# B&R Automation Studio project NAEUL004C00R13L518F00 (part 25)

#### Act_OptP1024Save.st
```iecst
ACTION Act_OptP1024Save:

	IF tyP1024McSetAntiGap.tyAntiGap.tyNumLftSenOff.bRtCompl
		OR tyP1024McSetAntiGap.tyAntiGap.tyNumMidSenOff.bRtCompl
		OR tyP1024McSetAntiGap.tyAntiGap.tyNumRgtSenOff.bRtCompl
		OR tyP1024McSetAntiGap.tyAntiGap.tyNumClrSenOff.bRtCompl
		OR tyP1024McSetAntiGap.tyAntiGap.tyNumMagConvEntOn.bRtCompl
		OR tyP1024McSetAntiGap.tyAntiGap.tyNumMagConvEntOff.bRtCompl
		OR tyP1024McSetAntiGap.tyAntiGap.tyNumMagConvPresentOn.bRtCompl
		OR tyP1024McSetAntiGap.tyAntiGap.tyNumMagConvPresentOff.bRtCompl
		THEN

		fUIInRtStatHide(ADR(tyCommon.tySet.tyBtnSave.uiMaskRtStat));

		tyP1024McSetAntiGap.tyAntiGap.tyNumLftSenOff.bRtCompl			:= FALSE;
		tyP1024McSetAntiGap.tyAntiGap.tyNumMidSenOff.bRtCompl			:= FALSE;
		tyP1024McSetAntiGap.tyAntiGap.tyNumRgtSenOff.bRtCompl			:= FALSE;
		tyP1024McSetAntiGap.tyAntiGap.tyNumClrSenOff.bRtCompl			:= FALSE;
		tyP1024McSetAntiGap.tyAntiGap.tyNumMagConvEntOn.bRtCompl		:= FALSE;
		tyP1024McSetAntiGap.tyAntiGap.tyNumMagConvEntOff.bRtCompl		:= FALSE;
		tyP1024McSetAntiGap.tyAntiGap.tyNumMagConvPresentOn.bRtCompl	:= FALSE;
		tyP1024McSetAntiGap.tyAntiGap.tyNumMagConvPresentOff.bRtCompl	:= FALSE;

	END_IF

	IF tyCommon.tySet.tyBtnSave.bRtCompl = TRUE THEN

		tyMcParamWr.tyLftSenAntiGapDly.diSigOffTm			:=  tyP1024McSetAntiGap.tyAntiGap.tyNumLftSenOff.diValue;
		tyMcParamWr.tyMidSenAntiGapDly.diSigOffTm			:=  tyP1024McSetAntiGap.tyAntiGap.tyNumMidSenOff.diValue;
		tyMcParamWr.tyRgtSenAntiGapDly.diSigOffTm			:=	tyP1024McSetAntiGap.tyAntiGap.tyNumRgtSenOff.diValue;
		tyMcParamWr.tyClrSenAntiGapDly.diSigOffTm			:=  tyP1024McSetAntiGap.tyAntiGap.tyNumClrSenOff.diValue;
		tyMcParamWr.tyMagConvEntrySenAntiGapDly.diSigOnTm	:=  tyP1024McSetAntiGap.tyAntiGap.tyNumMagConvEntOn.diValue;
		tyMcParamWr.tyMagConvEntrySenAntiGapDly.diSigOffTm	:=  tyP1024McSetAntiGap.tyAntiGap.tyNumMagConvEntOff.diValue;
		tyMcParamWr.tyMagConvPresentSenAntiGapDly.diSigOnTm	:=	tyP1024McSetAntiGap.tyAntiGap.tyNumMagConvPresentOn.diValue;
		tyMcParamWr.tyMagConvPresentSenAntiGapDly.diSigOffTm:=	tyP1024McSetAntiGap.tyAntiGap.tyNumMagConvPresentOff.diValue;

		eMcParamAct	:= McParamActWrite;

		IF p_eMcParamStat = McParamActWrite AND p_eMcParamStatus = Done THEN

			eMcParamAct	:= McParamActIdle;

			//Update BackUp Param
			tyP1024McSetAntiGap.tyAntiGapBkUp	:= tyP1024McSetAntiGap.tyAntiGap;

			tyCommon.tySet.tyBtnSave.bRtCompl 	:= FALSE;
			fUIInRtStatOff(ADR(tyCommon.tySet.tyBtnSave.uiMaskRtStat));

		ELSIF p_eMcParamStatus = Error THEN
			p_tyC0008MsgBox ACCESS ADR(tyP1024McSetAntiGap.tyMsgBoxSaveErr);

			IF tyP1024McSetAntiGap.tyMsgBoxSaveErr.tyBtnNo.bRtCompl = TRUE THEN
				tyP1024McSetAntiGap.tyMsgBoxSaveErr.tyBtnNo.bRtCompl	:= FALSE;
				tyP1024McSetAntiGap.tyMsgBoxSaveErr.tyBtnNo.bValue		:= FALSE;

				p_tyC0008MsgBox ACCESS ADR(tyP1024McSetAntiGap.tyMsgBoxHide);

				//Restore Param
				tyP1024McSetAntiGap.tyAntiGap	:= tyP1024McSetAntiGap.tyAntiGapBkUp;
				tyMcParamWr						:= p_tyMcParamCurr;

				tyCommon.tySet.tyBtnSave.bRtCompl 	:= FALSE;
				fUIInRtStatOff(ADR(tyCommon.tySet.tyBtnSave.uiMaskRtStat));
			END_IF

		END_IF

	END_IF

END_ACTION
```

#### Act_OptP1024Keypad.st
```iecst
ACTION Act_OptP1024Keypad:

	IF fUIOutRtStatTPIsOpen(ADR(tyP1024McSetAntiGap.tyAntiGap.tyNumLftSenOff.uiRtStat)) = TRUE THEN
		tyProperty.tyKeypad.tyStringTitle.sKeypadTitle	:= tyP1024McSetAntiGap.tyAntiGap.tyNumLftSenOff.sKeypadTitle;

	ELSIF fUIOutRtStatTPIsOpen(ADR(tyP1024McSetAntiGap.tyAntiGap.tyNumMidSenOff.uiRtStat)) = TRUE THEN
		tyProperty.tyKeypad.tyStringTitle.sKeypadTitle	:= tyP1024McSetAntiGap.tyAntiGap.tyNumMidSenOff.sKeypadTitle;

	ELSIF fUIOutRtStatTPIsOpen(ADR(tyP1024McSetAntiGap.tyAntiGap.tyNumRgtSenOff.uiRtStat)) = TRUE THEN
		tyProperty.tyKeypad.tyStringTitle.sKeypadTitle	:= tyP1024McSetAntiGap.tyAntiGap.tyNumRgtSenOff.sKeypadTitle;

	ELSIF fUIOutRtStatTPIsOpen(ADR(tyP1024McSetAntiGap.tyAntiGap.tyNumClrSenOff.uiRtStat)) = TRUE THEN
		tyProperty.tyKeypad.tyStringTitle.sKeypadTitle	:= tyP1024McSetAntiGap.tyAntiGap.tyNumClrSenOff.sKeypadTitle;

	ELSIF fUIOutRtStatTPIsOpen(ADR(tyP1024McSetAntiGap.tyAntiGap.tyNumMagConvEntOff.uiRtStat)) = TRUE THEN
		tyProperty.tyKeypad.tyStringTitle.sKeypadTitle	:= tyP1024McSetAntiGap.tyAntiGap.tyNumMagConvEntOff.sKeypadTitle;

	ELSIF fUIOutRtStatTPIsOpen(ADR(tyP1024McSetAntiGap.tyAntiGap.tyNumMagConvEntOn.uiRtStat)) = TRUE THEN
		tyProperty.tyKeypad.tyStringTitle.sKeypadTitle	:= tyP1024McSetAntiGap.tyAntiGap.tyNumMagConvEntOn.sKeypadTitle;

	ELSIF fUIOutRtStatTPIsOpen(ADR(tyP1024McSetAntiGap.tyAntiGap.tyNumMagConvPresentOff.uiRtStat)) = TRUE THEN
		tyProperty.tyKeypad.tyStringTitle.sKeypadTitle	:= tyP1024McSetAntiGap.tyAntiGap.tyNumMagConvEntOn.sKeypadTitle;

	ELSIF fUIOutRtStatTPIsOpen(ADR(tyP1024McSetAntiGap.tyAntiGap.tyNumMagConvPresentOn.uiRtStat)) = TRUE THEN
		tyProperty.tyKeypad.tyStringTitle.sKeypadTitle	:= tyP1024McSetAntiGap.tyAntiGap.tyNumMagConvEntOn.sKeypadTitle;

	END_IF

END_ACTION
```

#### Act_EntP1025Disp.st
```iecst
ACTION Act_EntP1025Disp:

	//Access Address
	p_tyC0004Navi ACCESS ADR(tyP1025McSetScan.tyNaviBack);

	p_tyC0005Main ACCESS ADR(tyCommon.tyMain);

	p_tyC0006Set ACCESS ADR(tyCommon.tySet);

	p_tyC0007Notif ACCESS ADR(tyCommon.tyNotif);

	p_tyC0008MsgBox ACCESS ADR (tyP1025McSetScan.tyMsgBoxHide);

	p_tyC0009Info ACCESS ADR(tyCommon.tyInfo);

	p_tyP1025McSetScan ACCESS ADR(tyP1025McSetScan.tyScan);

	//Backup Param
	tyP1025McSetScan.tyScanBkUp	:= tyP1025McSetScan.tyScan;

END_ACTION
```

#### Act_ExitP1025.st
```iecst
ACTION Act_ExitP1025:

	IF tyCommon.tySet.tyBtnSave.uiMaskRtStat.0 = FALSE THEN
		usiChgPage	:= 1;

	ELSE

		p_tyC0008MsgBox ACCESS ADR(tyP1025McSetScan.tyMsgBoxExitAsk);

		IF tyP1025McSetScan.tyMsgBoxExitAsk.tyBtnYes.bRtCompl = TRUE THEN
			tyP1025McSetScan.tyMsgBoxExitAsk.tyBtnYes.bRtCompl	:= FALSE;
			tyP1025McSetScan.tyMsgBoxExitAsk.tyBtnYes.bValue		:= FALSE;

			p_tyC0008MsgBox ACCESS ADR(tyP1025McSetScan.tyMsgBoxHide);

			//Restore Param
			tyP1025McSetScan.tyScan	:= tyP1025McSetScan.tyScanBkUp;

			fUIInRtStatOff(ADR(tyCommon.tySet.tyBtnSave.uiMaskRtStat));

			usiChgPage	:= 1;

		ELSIF tyP1025McSetScan.tyMsgBoxExitAsk.tyBtnNo.bRtCompl = TRUE THEN
			tyP1025McSetScan.tyMsgBoxExitAsk.tyBtnNo.bRtCompl	:= FALSE;
			tyP1025McSetScan.tyMsgBoxExitAsk.tyBtnNo.bValue		:= FALSE;

			p_tyC0008MsgBox ACCESS ADR(tyP1025McSetScan.tyMsgBoxHide);

			eChgPage	:= eCurrPage;
			usiChgPage	:= 0;

		END_IF

	END_IF

END_ACTION
```

#### Act_OptP1025Navi.st
```iecst
ACTION Act_OptP1025Navi:

	tyP1025McSetScan.tyNaviBack.tyBtnBack.bRtLk	:= tyCommon.tySet.tyBtnSave.bRtCompl;

	IF tyP1025McSetScan.tyNaviBack.tyBtnBack.bRtCompl = TRUE THEN
		tyP1025McSetScan.tyNaviBack.tyBtnBack.bRtCompl	:= FALSE;

		eChgPage	:= UIP1020McSetNavi;

	END_IF

END_ACTION
```

#### Act_OptP1025Save.st
```iecst
ACTION Act_OptP1025Save:

	IF tyP1025McSetScan.tyScan.tyStringTopScanSvrIP.bRtCompl OR tyP1025McSetScan.tyScan.tyNumTopScanSvrPort.bRtCompl
		OR tyP1025McSetScan.tyScan.tyStringTopScanSvrIP.bRtCompl OR tyP1025McSetScan.tyScan.tyNumBtmScanSvrPort.bRtCompl
		OR tyP1025McSetScan.tyScan.tyBtnTopScanEn.bRtCompl OR tyP1025McSetScan.tyScan.tyBtnBtmScanEn.bRtCompl THEN

		fUIInRtStatHide(ADR(tyCommon.tySet.tyBtnSave.uiMaskRtStat));

		tyP1025McSetScan.tyScan.tyStringTopScanSvrIP.bRtCompl			:= FALSE;
		tyP1025McSetScan.tyScan.tyNumTopScanSvrPort.bRtCompl			:= FALSE;
		tyP1025McSetScan.tyScan.tyStringTopScanSvrIP.bRtCompl			:= FALSE;
		tyP1025McSetScan.tyScan.tyNumBtmScanSvrPort.bRtCompl			:= FALSE;
		tyP1025McSetScan.tyScan.tyBtnTopScanEn.bRtCompl					:= FALSE;
		tyP1025McSetScan.tyScan.tyBtnBtmScanEn.bRtCompl					:= FALSE;

	END_IF

	IF tyCommon.tySet.tyBtnSave.bRtCompl = TRUE THEN

		tyMcParamWr.sTopScanIPAddr			:=  tyP1025McSetScan.tyScan.tyStringTopScanSvrIP.sValue;
		tyMcParamWr.uiTopScanSvrPort		:=  DINT_TO_UINT (tyP1025McSetScan.tyScan.tyNumTopScanSvrPort.diValue);
		tyMcParamWr.sBtmScanIPAddr			:=	tyP1025McSetScan.tyScan.tyStringBtmScanSvrIP.sValue;
		tyMcParamWr.uiBtmScanSvrPort		:=  DINT_TO_UINT (tyP1025McSetScan.tyScan.tyNumBtmScanSvrPort.diValue);
		tyMcParamWr.bTopScannerEn			:=  tyP1025McSetScan.tyScan.tyBtnTopScanEn.bValue;
		tyMcParamWr.bBtmScannerEn			:=  tyP1025McSetScan.tyScan.tyBtnBtmScanEn.bValue;

		eMcParamAct	:= McParamActWrite;

		IF p_eMcParamStat = McParamActWrite AND p_eMcParamStatus = Done THEN

			eMcParamAct	:= McParamActIdle;

			//Update BackUp Param
			tyP1025McSetScan.tyScanBkUp	:= tyP1025McSetScan.tyScan;

			tyCommon.tySet.tyBtnSave.bRtCompl 	:= FALSE;
			fUIInRtStatOff(ADR(tyCommon.tySet.tyBtnSave.uiMaskRtStat));

		ELSIF p_eMcParamStatus = Error THEN
			p_tyC0008MsgBox ACCESS ADR(tyP1025McSetScan.tyMsgBoxSaveErr);

			IF tyP1025McSetScan.tyMsgBoxSaveErr.tyBtnNo.bRtCompl = TRUE THEN
				tyP1025McSetScan.tyMsgBoxSaveErr.tyBtnNo.bRtCompl	:= FALSE;
				tyP1025McSetScan.tyMsgBoxSaveErr.tyBtnNo.bValue		:= FALSE;

				p_tyC0008MsgBox ACCESS ADR(tyP1025McSetScan.tyMsgBoxHide);

				//Restore Param
				tyP1025McSetScan.tyScan	:= tyP1025McSetScan.tyScanBkUp;
				tyMcParamWr						:= p_tyMcParamCurr;

				tyCommon.tySet.tyBtnSave.bRtCompl 	:= FALSE;
				fUIInRtStatOff(ADR(tyCommon.tySet.tyBtnSave.uiMaskRtStat));
			END_IF

		END_IF

	END_IF

END_ACTION
```

#### Act_OptP1025Keypad.st
```iecst
ACTION Act_OptP1025Keypad:

	IF fUIOutRtStatTPIsOpen(ADR(tyP1025McSetScan.tyScan.tyStringTopScanSvrIP.uiRtStat)) = TRUE THEN
		tyProperty.tyKeypad.tyStringTitle.sKeypadTitle	:= tyP1025McSetScan.tyScan.tyStringTopScanSvrIP.sKeypadTitle;

	ELSIF fUIOutRtStatTPIsOpen(ADR(tyP1025McSetScan.tyScan.tyNumTopScanSvrPort.uiRtStat)) = TRUE THEN
		tyProperty.tyKeypad.tyStringTitle.sKeypadTitle	:= tyP1025McSetScan.tyScan.tyNumTopScanSvrPort.sKeypadTitle;

	ELSIF fUIOutRtStatTPIsOpen(ADR(tyP1025McSetScan.tyScan.tyStringBtmScanSvrIP.uiRtStat)) = TRUE THEN
		tyProperty.tyKeypad.tyStringTitle.sKeypadTitle	:= tyP1025McSetScan.tyScan.tyStringBtmScanSvrIP.sKeypadTitle;

	ELSIF fUIOutRtStatTPIsOpen(ADR(tyP1025McSetScan.tyScan.tyNumBtmScanSvrPort.uiRtStat)) = TRUE THEN
		tyProperty.tyKeypad.tyStringTitle.sKeypadTitle	:= tyP1025McSetScan.tyScan.tyNumBtmScanSvrPort.sKeypadTitle;

	END_IF

END_ACTION
```

#### Act_EntP1026Disp.st
```iecst
ACTION Act_EntP1026Disp:

	//Access Address
	p_tyC0002FullMask ACCESS ADR(tyP1026McSetTeach.tyFullMaskHide);

	p_tyC0004Navi ACCESS ADR(tyP1026McSetTeach.tyNaviBack);

	p_tyC0005Main ACCESS ADR(tyCommon.tyMain);

	p_tyC0007Notif ACCESS ADR(tyCommon.tyNotif);

	p_tyC0008MsgBox ACCESS ADR(tyP1026McSetTeach.tyMsgBoxHide);

	p_tyC0009Info ACCESS ADR(tyCommon.tyInfo);

	p_tyP1026InOutletShutterFB ACCESS ADR(tyP1026McSetTeach.tyInOutletShutterFB);

	IF bTeachTravPosA = TRUE THEN
		p_tyP1026McSetTeach ACCESS ADR(tyP1026McSetTeach.tyTeachTravPosA);
		p_tyC0001MotionStd ACCESS ADR(tyP1026McSetTeach.tyMotionStdTrav);

	ELSIF bTeachTravPosB = TRUE THEN
		p_tyP1026McSetTeach ACCESS ADR(tyP1026McSetTeach.tyTeachTravPosB);
		p_tyC0001MotionStd ACCESS ADR(tyP1026McSetTeach.tyMotionStdTrav);

	ELSIF bTeachLifterPosA = TRUE THEN
		p_tyP1026McSetTeach ACCESS ADR(tyP1026McSetTeach.tyTeachLifterPosA);
		p_tyC0001MotionStd ACCESS ADR(tyP1026McSetTeach.tyMotionStdLifter);

	ELSIF bTeachLifterPosB = TRUE THEN
		p_tyP1026McSetTeach ACCESS ADR(tyP1026McSetTeach.tyTeachLifterPosB);
		p_tyC0001MotionStd ACCESS ADR(tyP1026McSetTeach.tyMotionStdLifter);

	ELSIF bTeachLifterTopPos THEN
		p_tyP1026McSetTeach ACCESS ADR(tyP1026McSetTeach.tyTeachLifterTopPos);
		p_tyC0001MotionStd ACCESS ADR(tyP1026McSetTeach.tyMotionStdLifter);

	ELSIF bTeachLifterBtmPos THEN
		p_tyP1026McSetTeach ACCESS ADR(tyP1026McSetTeach.tyTeachLifterBtmPos);
		p_tyC0001MotionStd ACCESS ADR(tyP1026McSetTeach.tyMotionStdLifter);

	ELSIF bTeachLifterTopPos2 THEN
		p_tyP1026McSetTeach ACCESS ADR(tyP1026McSetTeach.tyTeachLifterTopPos2);
		p_tyC0001MotionStd ACCESS ADR(tyP1026McSetTeach.tyMotionStdLifter); //Lifter2FBCtrl

	ELSIF bTeachLifterBtmPos2 THEN
		p_tyP1026McSetTeach ACCESS ADR(tyP1026McSetTeach.tyTeachLifterBtmPos2);
		p_tyC0001MotionStd ACCESS ADR(tyP1026McSetTeach.tyMotionStdLifter);

	END_IF

	//Display
	//Traverser
	tyP1026McSetTeach.tyMotionStdTrav.tyBtnPwr.bValue	:= p_bTravPwrOn;

	//Lifter
	tyP1026McSetTeach.tyMotionStdLifter.tyBtnPwr.bValue	:= p_bLifterBtmPwrOn;

END_ACTION
```

#### Act_ExitP1026.st
```iecst
ACTION Act_ExitP1026:

	usiChgPage	:= 1;

	//Manual Deactivated
	bManualMod	:= FALSE;

	//Reset UI
	bJogSlow				:= FALSE;
	bJogFast				:= FALSE;
	fbJogSlowToFastDlyTm.IN	:= FALSE;

	fbLmtRstTm(IN := FALSE);
	//bypass curtain sensor
	bBypCurtainSen := FALSE;
	bBypCurtainPBLED := FALSE;
	tyP1026McSetTeach.tyTeachTravPosA.tyBtn4.bValue				:= FALSE;
	tyP1026McSetTeach.tyTeachTravPosB.tyBtn4.bValue				:= FALSE;
	tyP1026McSetTeach.tyTeachLifterPosA.tyBtn4.bValue				:= FALSE;
	tyP1026McSetTeach.tyTeachLifterPosB.tyBtn4.bValue				:= FALSE;

	//Traverser
	tyP1026McSetTeach.tyMotionStdTrav.tyBtnPwr.bRtCompl				:= FALSE;
	tyP1026McSetTeach.tyMotionStdTrav.tyBtnStop.bRtCompl			:= FALSE;
	tyP1026McSetTeach.tyMotionStdTrav.tyBtnOrigin.bRtCompl			:= FALSE;
	tyP1026McSetTeach.tyMotionStdTrav.tyBtnRst.bRtCompl				:= FALSE;
	tyP1026McSetTeach.tyMotionStdTrav.tyBtnMovAbs.bRtCompl			:= FALSE;
	tyP1026McSetTeach.tyMotionStdTrav.tyBtnMovRel.bRtCompl			:= FALSE;
	tyP1026McSetTeach.tyMotionStdTrav.tyBtnJogFront.bRtCompl		:= FALSE;
	tyP1026McSetTeach.tyMotionStdTrav.tyBtnJogRear.bRtCompl			:= FALSE;

	tyP1026McSetTeach.tyTeachTravPosA.tyBtn2.bRtCompl				:= FALSE;
	tyP1026McSetTeach.tyTeachTravPosB.tyBtn2.bRtCompl				:= FALSE;

	tyP1026McSetTeach.tyMotionStdTrav.tyBtnPwr.bValue				:= FALSE;
	tyP1026McSetTeach.tyMotionStdTrav.tyBtnStop.bValue				:= TRUE;
	tyP1026McSetTeach.tyMotionStdTrav.tyBtnOrigin.bValue			:= FALSE;
	tyP1026McSetTeach.tyMotionStdTrav.tyBtnRst.bValue				:= FALSE;
	tyP1026McSetTeach.tyMotionStdTrav.tyBtnMovAbs.bValue			:= FALSE;
	tyP1026McSetTeach.tyMotionStdTrav.tyBtnMovRel.bValue			:= FALSE;
	tyP1026McSetTeach.tyMotionStdTrav.tyBtnJogFront.bValue			:= FALSE;
	tyP1026McSetTeach.tyMotionStdTrav.tyBtnJogRear.bValue			:= FALSE;

	tyP1026McSetTeach.tyTeachTravPosA.tyBtn2.bValue					:= FALSE;
	tyP1026McSetTeach.tyTeachTravPosB.tyBtn2.bValue					:= FALSE;

	tyP1026McSetTeach.tyMotionStdTrav.tyBtnPwr.bRtLk				:= FALSE;
	tyP1026McSetTeach.tyMotionStdTrav.tyBtnStop.bRtLk				:= TRUE;
	tyP1026McSetTeach.tyMotionStdTrav.tyBtnOrigin.bRtLk				:= FALSE;
	tyP1026McSetTeach.tyMotionStdTrav.tyBtnRst.bRtLk				:= FALSE;
	tyP1026McSetTeach.tyMotionStdTrav.tyBtnMovAbs.bRtLk				:= FALSE;
	tyP1026McSetTeach.tyMotionStdTrav.tyBtnMovRel.bRtLk				:= FALSE;
	tyP1026McSetTeach.tyMotionStdTrav.tyBtnJogFront.bRtLk			:= FALSE;
	tyP1026McSetTeach.tyMotionStdTrav.tyBtnJogRear.bRtLk			:= FALSE;

	tyP1026McSetTeach.tyTeachTravPosA.tyBtn2.bRtLk					:= FALSE;
	tyP1026McSetTeach.tyTeachTravPosB.tyBtn2.bRtLk					:= FALSE;

	tyP1026McSetTeach.tyMotionStdTrav.tyBtnPwr.uiMaskRtStat			:= TRUE;
	tyP1026McSetTeach.tyMotionStdTrav.tyBtnOrigin.uiMaskRtStat		:= FALSE;
	tyP1026McSetTeach.tyMotionStdTrav.tyBtnRst.uiMaskRtStat			:= TRUE;
	tyP1026McSetTeach.tyMotionStdTrav.tyBtnMovAbs.uiMaskRtStat		:= FALSE;
	tyP1026McSetTeach.tyMotionStdTrav.tyBtnMovRel.uiMaskRtStat		:= FALSE;
	tyP1026McSetTeach.tyMotionStdTrav.tyBtnJogFront.uiMaskRtStat	:= FALSE;
	tyP1026McSetTeach.tyMotionStdTrav.tyBtnJogRear.uiMaskRtStat		:= FALSE;

	tyP1026McSetTeach.tyTeachTravPosA.tyBtn2.uiMaskRtStat			:= FALSE;
	tyP1026McSetTeach.tyTeachTravPosB.tyBtn2.uiMaskRtStat			:= FALSE;

	//Lifter
	tyP1026McSetTeach.tyMotionStdLifter.tyBtnPwr.bRtCompl			:= FALSE;
	tyP1026McSetTeach.tyMotionStdLifter.tyBtnStop.bRtCompl			:= FALSE;
	tyP1026McSetTeach.tyMotionStdLifter.tyBtnOrigin.bRtCompl		:= FALSE;
	tyP1026McSetTeach.tyMotionStdLifter.tyBtnRst.bRtCompl			:= FALSE;
	tyP1026McSetTeach.tyMotionStdLifter.tyBtnMovAbs.bRtCompl		:= FALSE;
	tyP1026McSetTeach.tyMotionStdLifter.tyBtnMovRel.bRtCompl		:= FALSE;
	tyP1026McSetTeach.tyMotionStdLifter.tyBtnJogUp.bRtCompl			:= FALSE;
	tyP1026McSetTeach.tyMotionStdLifter.tyBtnJogDown.bRtCompl		:= FALSE;

	tyP1026McSetTeach.tyTeachLifterPosA.tyBtn2.bRtCompl				:= FALSE;
	tyP1026McSetTeach.tyTeachLifterPosB.tyBtn2.bRtCompl				:= FALSE;
	//Lifter top/bottom
	tyP1026McSetTeach.tyTeachLifterTopPos.tyBtn2.bRtCompl				:= FALSE;
	tyP1026McSetTeach.tyTeachLifterBtmPos.tyBtn2.bRtCompl				:= FALSE;
	tyP1026McSetTeach.tyTeachLifterTopPos2.tyBtn2.bRtCompl				:= FALSE;
	tyP1026McSetTeach.tyTeachLifterBtmPos2.tyBtn2.bRtCompl				:= FALSE;

	tyP1026McSetTeach.tyMotionStdLifter.tyBtnPwr.bValue				:= FALSE;
	tyP1026McSetTeach.tyMotionStdLifter.tyBtnStop.bValue			:= TRUE;
	tyP1026McSetTeach.tyMotionStdLifter.tyBtnOrigin.bValue			:= FALSE;
	tyP1026McSetTeach.tyMotionStdLifter.tyBtnRst.bValue				:= FALSE;
	tyP1026McSetTeach.tyMotionStdLifter.tyBtnMovAbs.bValue			:= FALSE;
	tyP1026McSetTeach.tyMotionStdLifter.tyBtnMovRel.bValue			:= FALSE;
	tyP1026McSetTeach.tyMotionStdLifter.tyBtnJogUp.bValue			:= FALSE;
	tyP1026McSetTeach.tyMotionStdLifter.tyBtnJogDown.bValue			:= FALSE;

	tyP1026McSetTeach.tyTeachLifterPosA.tyBtn2.bValue				:= FALSE;
	tyP1026McSetTeach.tyTeachLifterPosB.tyBtn2.bValue				:= FALSE;
	tyP1026McSetTeach.tyTeachLifterTopPos.tyBtn2.bValue				:= FALSE;
	tyP1026McSetTeach.tyTeachLifterBtmPos.tyBtn2.bValue				:= FALSE;
	tyP1026McSetTeach.tyTeachLifterTopPos2.tyBtn2.bValue				:= FALSE;
	tyP1026McSetTeach.tyTeachLifterBtmPos2.tyBtn2.bValue				:= FALSE;

	tyP1026McSetTeach.tyMotionStdLifter.tyBtnPwr.bRtLk				:= FALSE;
	tyP1026McSetTeach.tyMotionStdLifter.tyBtnStop.bRtLk				:= TRUE;
	tyP1026McSetTeach.tyMotionStdLifter.tyBtnOrigin.bRtLk			:= FALSE;
	tyP1026McSetTeach.tyMotionStdLifter.tyBtnRst.bRtLk				:= FALSE;
	tyP1026McSetTeach.tyMotionStdLifter.tyBtnMovAbs.bRtLk			:= FALSE;
	tyP1026McSetTeach.tyMotionStdLifter.tyBtnMovRel.bRtLk			:= FALSE;
	tyP1026McSetTeach.tyMotionStdLifter.tyBtnJogUp.bRtLk			:= FALSE;
	tyP1026McSetTeach.tyMotionStdLifter.tyBtnJogDown.bRtLk			:= FALSE;

	tyP1026McSetTeach.tyTeachLifterPosA.tyBtn2.bRtLk				:= FALSE;
	tyP1026McSetTeach.tyTeachLifterPosB.tyBtn2.bRtLk				:= FALSE;
	tyP1026McSetTeach.tyTeachLifterTopPos.tyBtn2.bRtLk				:= FALSE;
	tyP1026McSetTeach.tyTeachLifterBtmPos.tyBtn2.bRtLk				:= FALSE;
	tyP1026McSetTeach.tyTeachLifterTopPos2.tyBtn2.bRtLk				:= FALSE;
	tyP1026McSetTeach.tyTeachLifterBtmPos2.tyBtn2.bRtLk				:= FALSE;

	tyP1026McSetTeach.tyMotionStdLifter.tyBtnPwr.uiMaskRtStat		:= TRUE;
	tyP1026McSetTeach.tyMotionStdLifter.tyBtnOrigin.uiMaskRtStat	:= FALSE;
	tyP1026McSetTeach.tyMotionStdLifter.tyBtnRst.uiMaskRtStat		:= TRUE;
	tyP1026McSetTeach.tyMotionStdLifter.tyBtnMovAbs.uiMaskRtStat	:= FALSE;
	tyP1026McSetTeach.tyMotionStdLifter.tyBtnMovRel.uiMaskRtStat	:= FALSE;
	tyP1026McSetTeach.tyMotionStdLifter.tyBtnJogUp.uiMaskRtStat		:= FALSE;
	tyP1026McSetTeach.tyMotionStdLifter.tyBtnJogDown.uiMaskRtStat	:= FALSE;

	tyP1026McSetTeach.tyTeachLifterPosA.tyBtn2.uiMaskRtStat			:= FALSE;
	tyP1026McSetTeach.tyTeachLifterPosB.tyBtn2.uiMaskRtStat			:= FALSE;
	tyP1026McSetTeach.tyTeachLifterTopPos.tyBtn2.uiMaskRtStat			:= FALSE;
	tyP1026McSetTeach.tyTeachLifterBtmPos.tyBtn2.uiMaskRtStat			:= FALSE;
	tyP1026McSetTeach.tyTeachLifterTopPos2.tyBtn2.uiMaskRtStat			:= FALSE;
	tyP1026McSetTeach.tyTeachLifterBtmPos2.tyBtn2.uiMaskRtStat			:= FALSE;

END_ACTION
```

#### Act_OptP1026Navi.st
```iecst
ACTION Act_OptP1026Navi:

	IF tyP1026McSetTeach.tyNaviBack.tyBtnBack.bRtCompl = TRUE THEN
		tyP1026McSetTeach.tyNaviBack.tyBtnBack.bRtCompl	:= FALSE;
		tyP1026McSetTeach.tyNaviBack.tyBtnBack.bValue	:= FALSE;

		eChgPage	:= UIP1021McSetGen;
	END_IF

END_ACTION
```

#### Act_OptP1026FullMask.st
```iecst
ACTION Act_OptP1026FullMask:

	IF eCurrPage = UIP1026McSetTeach THEN

		IF p_tyDI.bEStopSig = FALSE THEN
			p_tyC0002FullMask ACCESS ADR(tyP1026McSetTeach.tyFullMaskEStop);

		ELSIF p_tyDI.bCoverSWSig = FALSE THEN
			p_tyC0002FullMask ACCESS ADR(tyP1026McSetTeach.tyFullMaskCWSig);

		ELSIF p_tyDI.bSafetyRlySig = FALSE THEN
			p_tyC0002FullMask ACCESS ADR(tyP1026McSetTeach.tyFullMaskSafetyRly);

		ELSIF (bTeachLifterPosA OR bTeachLifterPosB) AND (p_tyDI.bLifterSafetyLmtSW1 = FALSE OR p_tyDI.bLifterSafetyLmtSW2 = FALSE) THEN
			p_tyC0002FullMask ACCESS ADR(tyP1026McSetTeach.tyFullMaskSafetyLmtSW);

		ELSIF (bTeachLifterPosA OR bTeachLifterPosB) AND p_tyDI.bLifterTimingBeltSen = FALSE THEN
			p_tyC0002FullMask ACCESS ADR(tyP1026McSetTeach.tyFullMaskTimingBelt);

		ELSE
			p_tyC0002FullMask ACCESS ADR(tyP1026McSetTeach.tyFullMaskHide);

		END_IF

	END_IF

END_ACTION
```

#### Act_OptP1026Mnl.st
```iecst
ACTION Act_OptP1026Mnl:

	bManualMod	:= p_tyDI.bSafetyRlySig;

END_ACTION
```

#### Act_OptP1026TravTeach.st
```iecst
ACTION Act_OptP1026TravTeach:

	IF tyP1026McSetTeach.tyTeachTravPosA.tyBtn1.bRtCompl = TRUE THEN

		p_tyC0008MsgBox ACCESS ADR(tyP1026McSetTeach.tyMsgBoxUpdtTravPosA);
		IF tyP1026McSetTeach.tyMsgBoxUpdtTravPosA.tyBtnNo.bRtCompl THEN  //tyBtnYes
			tyP1026McSetTeach.tyMsgBoxUpdtTravPosA.tyBtnNo.bRtCompl	:= FALSE;
			tyP1026McSetTeach.tyMsgBoxUpdtTravPosA.tyBtnNo.bValue	:= FALSE;

			p_tyC0008MsgBox ACCESS ADR(tyP1026McSetTeach.tyMsgBoxHide);

			//Write Actual Position To Machine Settings
			tyP1021McSetGen.tyGen.tyNumTravPosLaneA.diValue 	:= p_diTravActualPos;
			tyP1021McSetGen.tyGen.tyNumTravPosLaneA.bRtCompl	:= TRUE;

			//Back To Machine Settings
			eChgPage	:= UIP1021McSetGen;

			fUIInRtStatHide(ADR(tyCommon.tySet.tyBtnSave.uiMaskRtStat));

			tyP1026McSetTeach.tyTeachTravPosA.tyBtn1.bRtCompl	:= FALSE;
			tyP1026McSetTeach.tyTeachTravPosA.tyBtn1.bValue		:= FALSE;
//		ELSIF tyP1026McSetTeach.tyMsgBoxUpdtTravPosA.tyBtnNo.bRtCompl THEN
//			tyP1026McSetTeach.tyMsgBoxUpdtTravPosA.tyBtnNo.bRtCompl	:= FALSE;
//			tyP1026McSetTeach.tyMsgBoxUpdtTravPosA.tyBtnNo.bValue	:= FALSE;
//
//			p_tyC0008MsgBox ACCESS ADR(tyP1026McSetTeach.tyMsgBoxHide);
//
//			//Back To Machine Settings
//			eChgPage	:= UIP1021McSetGen;
//
//			tyP1026McSetTeach.tyTeachTravPosA.tyBtn1.bRtCompl	:= FALSE;
//			tyP1026McSetTeach.tyTeachTravPosA.tyBtn1.bValue		:= FALSE;

		END_IF

	ELSIF tyP1026McSetTeach.tyTeachTravPosB.tyBtn1.bRtCompl = TRUE THEN

		p_tyC0008MsgBox ACCESS ADR(tyP1026McSetTeach.tyMsgBoxUpdtTravPosB);
		IF tyP1026McSetTeach.tyMsgBoxUpdtTravPosB.tyBtnNo.bRtCompl THEN
			tyP1026McSetTeach.tyMsgBoxUpdtTravPosB.tyBtnNo.bRtCompl := FALSE;
			tyP1026McSetTeach.tyMsgBoxUpdtTravPosB.tyBtnNo.bValue 	:= FALSE;

			p_tyC0008MsgBox ACCESS ADR(tyP1026McSetTeach.tyMsgBoxHide);
			//Back To Machine Settings
			eChgPage	:= UIP1021McSetGen;

			tyP1026McSetTeach.tyTeachTravPosB.tyBtn1.bRtCompl	:= FALSE;
			tyP1026McSetTeach.tyTeachTravPosB.tyBtn1.bValue		:= FALSE;
//		ELSIF tyP1026McSetTeach.tyMsgBoxUpdtTravPosB.tyBtnNo.bRtCompl THEN
//			tyP1026McSetTeach.tyMsgBoxUpdtTravPosB.tyBtnNo.bRtCompl := FALSE;
//			tyP1026McSetTeach.tyMsgBoxUpdtTravPosB.tyBtnNo.bValue 	:= FALSE;
//
//			p_tyC0008MsgBox ACCESS ADR(tyP1026McSetTeach.tyMsgBoxHide);
//
//			//Write Actual Position To Machine Settings
//			tyP1021McSetGen.tyGen.tyNumTravPosLaneB.diValue 	:= p_diTravActualPos;
//			tyP1021McSetGen.tyGen.tyNumTravPosLaneB.bRtCompl	:= TRUE;
//
//			//Back To Machine Settings
//			eChgPage	:= UIP1021McSetGen;
//
//			fUIInRtStatHide(ADR(tyCommon.tySet.tyBtnSave.uiMaskRtStat));
//
//			tyP1026McSetTeach.tyTeachTravPosB.tyBtn1.bRtCompl	:= FALSE;
//			tyP1026McSetTeach.tyTeachTravPosB.tyBtn1.bValue		:= FALSE;

		END_IF

	END_IF

END_ACTION
```

#### Act_OptP1026TravFBCtrl.st
```iecst
ACTION Act_OptP1026TravFBCtrl:

	fbJogSlowToFastDlyTm.PT			:= T#2s;
	fbJogSlowToFastDlyTm;
	fbLmtRstTm;

//	IF EDGEPOS((p_udiTravAxisErrID = 21570 OR p_udiTravAxisErrID = 21571)
	IF EDGEPOS((p_bTravFwdLmtSen OR p_bTravRevLmtSen OR p_udiTravAxisErrID = 21570 OR p_udiTravAxisErrID = 21571)
		AND tyP1026McSetTeach.tyMotionStdTrav.tyBtnJogRear.bValue = FALSE
		AND tyP1026McSetTeach.tyMotionStdTrav.tyBtnJogFront.bValue = FALSE) THEN

		fbLmtRstTm.IN				:= TRUE;
	END_IF

	IF fbLmtRstTm.Q = TRUE THEN
		tyP1026McSetTeach.tyMotionStdTrav.tyBtnRst.bRtCompl		:= TRUE;
	END_IF

	IF (tyP1026McSetTeach.tyMotionStdTrav.tyBtnJogFront.bValue = FALSE AND tyP1026McSetTeach.tyMotionStdTrav.tyBtnJogRear.bValue = FALSE) AND (p_bTravJogging = TRUE) THEN
		bJogStopTrav	:= TRUE;
	END_IF

	IF tyP1026McSetTeach.tyMotionStdTrav.tyBtnStop.bRtCompl = TRUE THEN
		eTravAct		:= TravActStop;

		IF p_eTravStat = TravActStop AND p_eTravStatus = Done THEN
			eTravAct	:= TravActIdle;

			tyP1026McSetTeach.tyMotionStdTrav.tyBtnStop.bRtCompl		:= FALSE;
			tyP1026McSetTeach.tyMotionStdTrav.tyBtnJogRear.bRtCompl		:= FALSE;
			tyP1026McSetTeach.tyMotionStdTrav.tyBtnJogFront.bRtCompl	:= FALSE;
			tyP1026McSetTeach.tyMotionStdTrav.tyBtnOrigin.bRtCompl		:= FALSE;
			tyP1026McSetTeach.tyMotionStdTrav.tyBtnMovAbs.bRtCompl		:= FALSE;
			tyP1026McSetTeach.tyMotionStdTrav.tyBtnMovRel.bRtCompl		:= FALSE;

			tyP1026McSetTeach.tyTeachTravPosA.tyBtn2.bRtCompl			:= FALSE;
			tyP1026McSetTeach.tyTeachTravPosB.tyBtn2.bRtCompl			:= FALSE;

			tyP1026McSetTeach.tyMotionStdTrav.tyBtnStop.bValue			:= TRUE;
			tyP1026McSetTeach.tyMotionStdTrav.tyBtnJogRear.bValue		:= FALSE;
			tyP1026McSetTeach.tyMotionStdTrav.tyBtnJogFront.bValue		:= FALSE;
			tyP1026McSetTeach.tyMotionStdTrav.tyBtnOrigin.bValue		:= FALSE;
			tyP1026McSetTeach.tyMotionStdTrav.tyBtnMovAbs.bValue		:= FALSE;
			tyP1026McSetTeach.tyMotionStdTrav.tyBtnMovRel.bValue		:= FALSE;
			tyP1026McSetTeach.tyTeachTravPosA.tyBtn2.bValue				:= FALSE;
			tyP1026McSetTeach.tyTeachTravPosB.tyBtn2.bValue				:= FALSE;

			tyP1026McSetTeach.tyMotionStdTrav.tyBtnStop.bRtLk			:= TRUE;
			tyP1026McSetTeach.tyMotionStdTrav.tyBtnJogRear.bRtLk		:= FALSE;
			tyP1026McSetTeach.tyMotionStdTrav.tyBtnJogFront.bRtLk		:= FALSE;
			tyP1026McSetTeach.tyMotionStdTrav.tyBtnOrigin.bRtLk			:= FALSE;
			tyP1026McSetTeach.tyMotionStdTrav.tyBtnMovAbs.bRtLk			:= FALSE;
			tyP1026McSetTeach.tyMotionStdTrav.tyBtnMovRel.bRtLk			:= FALSE;

			tyP1026McSetTeach.tyTeachTravPosA.tyBtn2.bRtLk						:= FALSE;
			tyP1026McSetTeach.tyTeachTravPosB.tyBtn2.bRtLk						:= FALSE;
		END_IF

	ELSIF (tyP1026McSetTeach.tyMotionStdTrav.tyBtnJogRear.bRtCompl = TRUE) OR (tyP1026McSetTeach.tyMotionStdTrav.tyBtnJogFront.bRtCompl = TRUE) OR (bJogStopTrav = TRUE) THEN
		bJogSlow					:= FALSE;
		bJogFast					:= FALSE;
		fbJogSlowToFastDlyTm.IN		:= FALSE;

		eTravAct		:= TravActJogStop;

		IF p_eTravStat = TravActJogStop AND p_eTravStatus = Done THEN
			eTravAct		:= TravActIdle;

			bJogStopTrav	:= FALSE;

			tyP1026McSetTeach.tyMotionStdTrav.tyBtnStop.bRtCompl		:= FALSE;
			tyP1026McSetTeach.tyMotionStdTrav.tyBtnJogRear.bRtCompl		:= FALSE;
			tyP1026McSetTeach.tyMotionStdTrav.tyBtnJogFront.bRtCompl	:= FALSE;
			tyP1026McSetTeach.tyMotionStdTrav.tyBtnOrigin.bRtCompl		:= FALSE;
			tyP1026McSetTeach.tyMotionStdTrav.tyBtnMovAbs.bRtCompl		:= FALSE;
			tyP1026McSetTeach.tyMotionStdTrav.tyBtnMovRel.bRtCompl		:= FALSE;
			tyP1026McSetTeach.tyTeachTravPosA.tyBtn2.bRtCompl			:= FALSE;
			tyP1026McSetTeach.tyTeachTravPosB.tyBtn2.bRtCompl			:= FALSE;

			tyP1026McSetTeach.tyMotionStdTrav.tyBtnStop.bValue			:= TRUE;
			tyP1026McSetTeach.tyMotionStdTrav.tyBtnJogRear.bValue		:= FALSE;
			tyP1026McSetTeach.tyMotionStdTrav.tyBtnJogFront.bValue		:= FALSE;
			tyP1026McSetTeach.tyMotionStdTrav.tyBtnOrigin.bValue		:= FALSE;
			tyP1026McSetTeach.tyMotionStdTrav.tyBtnMovAbs.bValue		:= FALSE;
			tyP1026McSetTeach.tyMotionStdTrav.tyBtnMovRel.bValue		:= FALSE;
			tyP1026McSetTeach.tyTeachTravPosA.tyBtn2.bValue				:= FALSE;
			tyP1026McSetTeach.tyTeachTravPosB.tyBtn2.bValue				:= FALSE;

			tyP1026McSetTeach.tyMotionStdTrav.tyBtnStop.bRtLk			:= TRUE;
			tyP1026McSetTeach.tyMotionStdTrav.tyBtnJogRear.bRtLk		:= FALSE;
			tyP1026McSetTeach.tyMotionStdTrav.tyBtnJogFront.bRtLk		:= FALSE;
			tyP1026McSetTeach.tyMotionStdTrav.tyBtnOrigin.bRtLk			:= FALSE;
			tyP1026McSetTeach.tyMotionStdTrav.tyBtnMovAbs.bRtLk			:= FALSE;
			tyP1026McSetTeach.tyMotionStdTrav.tyBtnMovRel.bRtLk			:= FALSE;
			tyP1026McSetTeach.tyTeachTravPosA.tyBtn2.bRtLk				:= FALSE;
			tyP1026McSetTeach.tyTeachTravPosB.tyBtn2.bRtLk				:= FALSE;
		END_IF

	ELSIF tyP1026McSetTeach.tyMotionStdTrav.tyBtnPwr.bRtCompl = TRUE THEN
		tyP1026McSetTeach.tyMotionStdTrav.tyBtnPwr.bRtLk				:= TRUE;

		IF tyP1026McSetTeach.tyMotionStdTrav.tyBtnPwr.bValue = TRUE THEN
			eTravAct		:= TravActPwrOn;

			IF p_eTravStat = TravActPwrOn AND p_eTravStatus = Done THEN
				eTravAct	:= TravActIdle;

				tyP1026McSetTeach.tyMotionStdTrav.tyBtnPwr.bRtCompl		:= FALSE;
				tyP1026McSetTeach.tyMotionStdTrav.tyBtnPwr.bRtLk		:= FALSE;
			END_IF
		ELSE
			eTravAct		:= TravActPwrOff;

			IF p_eTravStat = TravActPwrOff AND p_eTravStatus = Done THEN
				eTravAct	:= TravActIdle;

				tyP1026McSetTeach.tyMotionStdTrav.tyBtnPwr.bRtCompl		:= FALSE;
				tyP1026McSetTeach.tyMotionStdTrav.tyBtnPwr.bRtLk		:= FALSE;
			END_IF
		END_IF

	ELSIF tyP1026McSetTeach.tyMotionStdTrav.tyBtnOrigin.bRtCompl = TRUE THEN
		tyP1026McSetTeach.tyMotionStdTrav.tyBtnOrigin.bValue			:= TRUE;
		tyP1026McSetTeach.tyMotionStdTrav.tyBtnStop.bValue				:= FALSE;

		tyP1026McSetTeach.tyMotionStdTrav.tyBtnOrigin.bRtLk				:= TRUE;
		tyP1026McSetTeach.tyMotionStdTrav.tyBtnStop.bRtLk				:= FALSE;

		eTravAct		:= TravActHoming;

		IF p_eTravStat = TravActHoming AND p_eTravStatus = Done THEN
			eTravAct	:= TravActIdle;

			tyP1026McSetTeach.tyMotionStdTrav.tyBtnOrigin.bRtCompl		:= FALSE;
			tyP1026McSetTeach.tyMotionStdTrav.tyBtnOrigin.bValue		:= FALSE;
			tyP1026McSetTeach.tyMotionStdTrav.tyBtnStop.bValue			:= TRUE;

			tyP1026McSetTeach.tyMotionStdTrav.tyBtnOrigin.bRtLk			:= FALSE;
			tyP1026McSetTeach.tyMotionStdTrav.tyBtnStop.bRtLk			:= TRUE;
		END_IF

	ELSIF tyP1026McSetTeach.tyMotionStdTrav.tyBtnRst.bRtCompl = TRUE THEN
		tyP1026McSetTeach.tyMotionStdTrav.tyBtnRst.bValue				:= TRUE;
		tyP1026McSetTeach.tyMotionStdTrav.tyBtnRst.bRtLk				:= TRUE;

		eTravAct		:= TravActRstAxisErr;

		IF p_eTravStat = TravActRstAxisErr AND p_eTravStatus = Done THEN
			eTravAct	:= TravActIdle;

			tyP1026McSetTeach.tyMotionStdTrav.tyBtnRst.bRtCompl			:= FALSE;
			tyP1026McSetTeach.tyMotionStdTrav.tyBtnRst.bValue			:= FALSE;
			tyP1026McSetTeach.tyMotionStdTrav.tyBtnRst.bRtLk			:= FALSE;

			fbLmtRstTm.IN			:= FALSE;
		END_IF

	ELSIF tyP1026McSetTeach.tyTeachTravPosA.tyBtn2.bRtCompl = TRUE THEN
		tyP1026McSetTeach.tyTeachTravPosA.tyBtn2.bValue		:= TRUE;
		tyP1026McSetTeach.tyMotionStdTrav.tyBtnStop.bValue	:= FALSE;

		tyP1026McSetTeach.tyTeachTravPosA.tyBtn2.bRtLk		:= TRUE;
		tyP1026McSetTeach.tyMotionStdTrav.tyBtnStop.bRtLk	:= FALSE;

		diMnlTravNomSpd	:= tyP1026McSetTeach.tyMotionStdTrav.tyNumNomSpd.diValue;

		eTravAct		:= TravActGoAPos;

		IF p_eTravStat = TravActGoAPos AND p_eTravStatus = Done THEN
			eTravAct	:= TravActIdle;

			tyP1026McSetTeach.tyTeachTravPosA.tyBtn2.bRtCompl	:= FALSE;
			tyP1026McSetTeach.tyTeachTravPosA.tyBtn2.bValue		:= FALSE;
			tyP1026McSetTeach.tyMotionStdTrav.tyBtnStop.bValue	:= TRUE;

			tyP1026McSetTeach.tyTeachTravPosA.tyBtn2.bRtLk		:= FALSE;
			tyP1026McSetTeach.tyMotionStdTrav.tyBtnStop.bRtLk	:= TRUE;
		END_IF

	ELSIF tyP1026McSetTeach.tyTeachTravPosB.tyBtn2.bRtCompl = TRUE THEN
		tyP1026McSetTeach.tyTeachTravPosB.tyBtn2.bValue		:= TRUE;
		tyP1026McSetTeach.tyMotionStdTrav.tyBtnStop.bValue	:= FALSE;

		tyP1026McSetTeach.tyTeachTravPosB.tyBtn2.bRtLk		:= TRUE;
		tyP1026McSetTeach.tyMotionStdTrav.tyBtnStop.bRtLk	:= FALSE;

		diMnlTravNomSpd	:= tyP1026McSetTeach.tyMotionStdTrav.tyNumNomSpd.diValue;

		eTravAct		:= TravActGoBPos;

		IF p_eTravStat = TravActGoBPos AND p_eTravStatus = Done THEN
			eTravAct	:= TravActIdle;

			tyP1026McSetTeach.tyTeachTravPosB.tyBtn2.bRtCompl	:= FALSE;
			tyP1026McSetTeach.tyTeachTravPosB.tyBtn2.bValue		:= FALSE;
			tyP1026McSetTeach.tyMotionStdTrav.tyBtnStop.bValue	:= TRUE;

			tyP1026McSetTeach.tyTeachTravPosB.tyBtn2.bRtLk		:= FALSE;
			tyP1026McSetTeach.tyMotionStdTrav.tyBtnStop.bRtLk	:= TRUE;
		END_IF

	ELSIF tyP1026McSetTeach.tyMotionStdTrav.tyBtnMovAbs.bRtCompl = TRUE THEN
		tyP1026McSetTeach.tyMotionStdTrav.tyBtnMovAbs.bValue	:= TRUE;
		tyP1026McSetTeach.tyMotionStdTrav.tyBtnStop.bValue		:= FALSE;

		tyP1026McSetTeach.tyMotionStdTrav.tyBtnMovAbs.bRtLk		:= TRUE;
		tyP1026McSetTeach.tyMotionStdTrav.tyBtnStop.bRtLk		:= FALSE;

		diMnlTravTargetPos	:= tyP1026McSetTeach.tyMotionStdTrav.tyNumTargetPos.diValue;
		diMnlTravNomSpd		:= tyP1026McSetTeach.tyMotionStdTrav.tyNumNomSpd.diValue;

		eTravAct		:= TravActMovAbs;

		IF p_eTravStat = TravActMovAbs AND p_eTravStatus = Done THEN
			eTravAct	:= TravActIdle;

			tyP1026McSetTeach.tyMotionStdTrav.tyBtnMovAbs.bRtCompl		:= FALSE;
			tyP1026McSetTeach.tyMotionStdTrav.tyBtnMovAbs.bValue		:= FALSE;
			tyP1026McSetTeach.tyMotionStdTrav.tyBtnStop.bValue			:= TRUE;

			tyP1026McSetTeach.tyMotionStdTrav.tyBtnMovAbs.bRtLk			:= FALSE;
			tyP1026McSetTeach.tyMotionStdTrav.tyBtnStop.bRtLk			:= TRUE;
		END_IF

	ELSIF tyP1026McSetTeach.tyMotionStdTrav.tyBtnMovRel.bRtCompl = TRUE THEN
		tyP1026McSetTeach.tyMotionStdTrav.tyBtnMovRel.bValue			:= TRUE;
		tyP1026McSetTeach.tyMotionStdTrav.tyBtnStop.bValue				:= FALSE;

		tyP1026McSetTeach.tyMotionStdTrav.tyBtnMovRel.bRtLk				:= TRUE;
		tyP1026McSetTeach.tyMotionStdTrav.tyBtnStop.bRtLk				:= FALSE;

		diMnlTravStepSize	:= tyP1026McSetTeach.tyMotionStdTrav.tyNumStepSize.diValue;
		diMnlTravNomSpd		:= tyP1026McSetTeach.tyMotionStdTrav.tyNumNomSpd.diValue;

		eTravAct		:= TravActMovRel;

		IF p_eTravStat = TravActMovRel AND p_eTravStatus = Done THEN
			eTravAct	:= TravActIdle;

			tyP1026McSetTeach.tyMotionStdTrav.tyBtnMovRel.bRtCompl		:= FALSE;
			tyP1026McSetTeach.tyMotionStdTrav.tyBtnMovRel.bValue		:= FALSE;
			tyP1026McSetTeach.tyMotionStdTrav.tyBtnStop.bValue			:= TRUE;

			tyP1026McSetTeach.tyMotionStdTrav.tyBtnMovRel.bRtLk			:= FALSE;
			tyP1026McSetTeach.tyMotionStdTrav.tyBtnStop.bRtLk			:= TRUE;
		END_IF

	ELSIF (tyP1026McSetTeach.tyMotionStdTrav.tyBtnJogRear.bValue = TRUE) AND (fbJogSlowToFastDlyTm.Q = FALSE) AND (bJogSlow = FALSE) THEN
		tyP1026McSetTeach.tyMotionStdTrav.tyBtnStop.bValue				:= FALSE;
		tyP1026McSetTeach.tyMotionStdTrav.tyBtnStop.bRtLk				:= FALSE;

		fbJogSlowToFastDlyTm.IN		:= TRUE;

		diMnlTravJogSpd	:= tyP1026McSetTeach.tyMotionStdTrav.tyNumSlwSpd.diValue;

		eTravAct		:= TravActJogRear;

		IF p_eTravStat = TravActJogRear AND p_eTravStatus = Done THEN
			eTravAct	:= TravActIdle;
			bJogSlow				:= TRUE;
		ELSIF p_eTravStatus = Error THEN
			fbJogSlowToFastDlyTm.IN	:= FALSE;
			bJogSlow				:= TRUE;
		END_IF

	ELSIF (tyP1026McSetTeach.tyMotionStdTrav.tyBtnJogRear.bValue = TRUE) AND (fbJogSlowToFastDlyTm.Q = TRUE) AND (bJogFast = FALSE) THEN
		tyP1026McSetTeach.tyMotionStdTrav.tyBtnStop.bValue					:= FALSE;
		tyP1026McSetTeach.tyMotionStdTrav.tyBtnStop.bRtLk					:= FALSE;

		fbJogSlowToFastDlyTm.IN		:= TRUE;

		diMnlTravJogSpd	:= tyP1026McSetTeach.tyMotionStdTrav.tyNumNomSpd.diValue;

		eTravAct		:= TravActJogRear;

		IF p_eTravStat = TravActJogRear AND p_eTravStatus = Done THEN
			eTravAct	:= TravActIdle;
			bJogFast				:= TRUE;
		ELSIF p_eTravStatus = Error THEN
			fbJogSlowToFastDlyTm.IN	:= FALSE;
			bJogFast				:= TRUE;
		END_IF

	ELSIF (tyP1026McSetTeach.tyMotionStdTrav.tyBtnJogFront.bValue = TRUE) AND (fbJogSlowToFastDlyTm.Q = FALSE) AND (bJogSlow = FALSE) THEN
		tyP1026McSetTeach.tyMotionStdTrav.tyBtnStop.bValue				:= FALSE;
		tyP1026McSetTeach.tyMotionStdTrav.tyBtnStop.bRtLk				:= FALSE;

		fbJogSlowToFastDlyTm.IN		:= TRUE;

		diMnlTravJogSpd	:= tyP1026McSetTeach.tyMotionStdTrav.tyNumSlwSpd.diValue;

		eTravAct		:= TravActJogFront;

		IF p_eTravStat = TravActJogFront AND p_eTravStatus = Done THEN
			eTravAct	:= TravActIdle;
			bJogSlow				:= TRUE;
		ELSIF p_eTravStatus = Error THEN
			fbJogSlowToFastDlyTm.IN	:= FALSE;
			bJogSlow				:= TRUE;
		END_IF

	ELSIF (tyP1026McSetTeach.tyMotionStdTrav.tyBtnJogFront.bValue = TRUE) AND (fbJogSlowToFastDlyTm.Q = TRUE) AND (bJogFast = FALSE) THEN
		tyP1026McSetTeach.tyMotionStdTrav.tyBtnStop.bValue				:= FALSE;
		tyP1026McSetTeach.tyMotionStdTrav.tyBtnStop.bRtLk				:= FALSE;

		fbJogSlowToFastDlyTm.IN		:= TRUE;

		diMnlTravJogSpd	:= tyP1026McSetTeach.tyMotionStdTrav.tyNumNomSpd.diValue;

		eTravAct		:= TravActJogFront;

		IF p_eTravStat = TravActJogFront AND p_eTravStatus = Done THEN
			eTravAct	:= TravActIdle;
			bJogFast	:= TRUE;
		ELSIF p_eTravStatus = Error THEN
			fbJogSlowToFastDlyTm.IN	:= FALSE;
			bJogFast				:= TRUE;
		END_IF
	END_IF

	IF tyP1026McSetTeach.tyInOutletShutterFB.tyBtnOpen.bRtCompl = TRUE THEN
		tyP1026McSetTeach.tyInOutletShutterFB.tyBtnOpen.bRtCompl	:= FALSE;

		tyP1026McSetTeach.tyInOutletShutterFB.tyBtnOpen.bValue	:= TRUE;
		tyP1026McSetTeach.tyInOutletShutterFB.tyBtnClose.bValue	:= FALSE;

	ELSIF tyP1026McSetTeach.tyInOutletShutterFB.tyBtnClose.bRtCompl = TRUE THEN
		tyP1026McSetTeach.tyInOutletShutterFB.tyBtnClose.bRtCompl	:= FALSE;

		tyP1026McSetTeach.tyInOutletShutterFB.tyBtnClose.bValue	:= TRUE;
		tyP1026McSetTeach.tyInOutletShutterFB.tyBtnOpen.bValue	:= FALSE;
	END_IF

	IF tyP1026McSetTeach.tyInOutletShutterFB.tyBtnOpen.bValue = TRUE THEN
		eInShutterAct	:= PneuActRet;
		eOutShutterAct	:= PneuActRet;
		eOutShutterAct2	:= PneuActRet;
		eOutShutterAct3	:= PneuActRet;

		IF (p_eInShutterStat = PneuActRet AND p_eInShutterStatus = Done)
			AND (p_eOutShutterStat = PneuActRet AND p_eOutShutterStatus = Done)
			AND (p_eOutShutterStat2 = PneuActRet AND p_eOutShutterStatus2 = Done)
			AND (p_eOutShutterStat3 = PneuActRet AND p_eOutShutterStatus3 = Done)
			THEN
			eInShutterAct	:= PneuActIdle;
			eOutShutterAct	:= PneuActIdle;
			eOutShutterAct2	:= PneuActIdle;
			eOutShutterAct3	:= PneuActIdle;
			tyP1026McSetTeach.tyInOutletShutterFB.tyBtnOpen.bValue	:= FALSE;
		ELSIF p_eInShutterStatus = Error OR p_eOutShutterStatus = Error OR p_eOutShutterStatus2 = Error OR p_eOutShutterStatus3 = Error THEN
			tyP1026McSetTeach.tyInOutletShutterFB.tyBtnOpen.bValue	:= FALSE;
		END_IF

	ELSIF tyP1026McSetTeach.tyInOutletShutterFB.tyBtnClose.bValue = TRUE THEN
		eInShutterAct	:= PneuActExt;
		eOutShutterAct	:= PneuActExt;
		eOutShutterAct2	:= PneuActExt;
		eOutShutterAct3	:= PneuActExt;
		IF (p_eInShutterStat = PneuActExt AND p_eInShutterStatus = Done)
			AND (p_eOutShutterStat = PneuActExt AND p_eOutShutterStatus = Done)
			AND (p_eOutShutterStat2 = PneuActExt AND p_eOutShutterStatus2 = Done)
			AND (p_eOutShutterStat3 = PneuActExt AND p_eOutShutterStatus3 = Done)
			THEN
			eInShutterAct	:= PneuActIdle;
			eOutShutterAct	:= PneuActIdle;
			eOutShutterAct2	:= PneuActIdle;
			eOutShutterAct3	:= PneuActIdle;
			tyP1026McSetTeach.tyInOutletShutterFB.tyBtnClose.bValue := FALSE;
		ELSIF p_eInShutterStatus = Error OR p_eOutShutterStatus = Error THEN
			tyP1026McSetTeach.tyInOutletShutterFB.tyBtnClose.bValue := FALSE;
		END_IF
	END_IF

	IF p_eTravStat = TravActJogStop AND (p_eTravStatus = Done OR p_eTravStatus = Error) THEN
		eTravAct		:= TravActIdle;
	END_IF

	//bypass curtain sensor
	IF bTeachTravPosA OR bTeachTravPosB THEN
		bBypCurtainSen			:= tyP1026McSetTeach.tyTeachTravPosA.tyBtn4.bValue OR tyP1026McSetTeach.tyTeachTravPosB.tyBtn4.bValue;
		bBypCurtainPBLED		:= tyP1026McSetTeach.tyTeachTravPosA.tyBtn4.bValue OR tyP1026McSetTeach.tyTeachTravPosB.tyBtn4.bValue;
	END_IF

END_ACTION
```

#### Act_OptP1026TravFBStat.st
```iecst
ACTION Act_OptP1026TravFBStat:

	IF p_bTravAxisErr = TRUE THEN
		tyP1026McSetTeach.tyMotionStdTrav.tyStringStat.sValue		:= p_sTravAxisErrTxt;
	ELSE
		tyP1026McSetTeach.tyMotionStdTrav.tyStringStat.sValue		:= p_sTravStatTxt;
	END_IF

END_ACTION
```

#### Act_OptP1026TravMask.st
```iecst
ACTION Act_OptP1026TravMask:

	// Interlock Power
	IF p_bTravAxisErr = TRUE AND p_bTravPwrOn = FALSE THEN
		fUIInRtStatOff(ADR(tyP1026McSetTeach.tyMotionStdTrav.tyBtnPwr.uiMaskRtStat));
		tyP1026McSetTeach.tyMotionStdTrav.tyBtnPwr.bValue		:= FALSE;
	ELSE
		fUIInRtStatHide(ADR(tyP1026McSetTeach.tyMotionStdTrav.tyBtnPwr.uiMaskRtStat));
	END_IF

	// Interlock Others Move
	IF p_bTravAxisErr = TRUE OR p_bTravPwrOn = FALSE THEN
		fUIInRtStatOff(ADR(tyP1026McSetTeach.tyMotionStdTrav.tyBtnOrigin.uiMaskRtStat));
		fUIInRtStatOff(ADR(tyP1026McSetTeach.tyMotionStdTrav.tyBtnMovRel.uiMaskRtStat));
		fUIInRtStatOff(ADR(tyP1026McSetTeach.tyMotionStdTrav.tyBtnJogFront.uiMaskRtStat));
		fUIInRtStatOff(ADR(tyP1026McSetTeach.tyMotionStdTrav.tyBtnJogRear.uiMaskRtStat));
	ELSE
		fUIInRtStatHide(ADR(tyP1026McSetTeach.tyMotionStdTrav.tyBtnOrigin.uiMaskRtStat));
		fUIInRtStatHide(ADR(tyP1026McSetTeach.tyMotionStdTrav.tyBtnMovRel.uiMaskRtStat));
		fUIInRtStatHide(ADR(tyP1026McSetTeach.tyMotionStdTrav.tyBtnJogFront.uiMaskRtStat));
		fUIInRtStatHide(ADR(tyP1026McSetTeach.tyMotionStdTrav.tyBtnJogRear.uiMaskRtStat));
	END_IF

	// Interlock Move Absolute
	IF p_bTravAxisErr = TRUE OR p_bTravPwrOn = FALSE OR p_bTravIsHomed = FALSE THEN
		fUIInRtStatOff(ADR(tyP1026McSetTeach.tyTeachTravPosA.tyBtn2.uiMaskRtStat));
		fUIInRtStatOff(ADR(tyP1026McSetTeach.tyTeachTravPosB.tyBtn2.uiMaskRtStat));
		fUIInRtStatOff(ADR(tyP1026McSetTeach.tyMotionStdTrav.tyBtnMovAbs.uiMaskRtStat));
	ELSE
		fUIInRtStatHide(ADR(tyP1026McSetTeach.tyTeachTravPosA.tyBtn2.uiMaskRtStat));
		fUIInRtStatHide(ADR(tyP1026McSetTeach.tyTeachTravPosB.tyBtn2.uiMaskRtStat));
		fUIInRtStatHide(ADR(tyP1026McSetTeach.tyMotionStdTrav.tyBtnMovAbs.uiMaskRtStat));
	END_IF

	//Interlock Limit Sensor
	IF tyP1026McSetTeach.tyMotionStdTrav.tyBtnRearLmtSen.bValue = TRUE THEN
		fUIInRtStatOff(ADR(tyP1026McSetTeach.tyMotionStdTrav.tyBtnJogRear.uiMaskRtStat));
	END_IF

	IF tyP1026McSetTeach.tyMotionStdTrav.tyBtnFrontLmtSen.bValue = TRUE THEN
		fUIInRtStatOff(ADR(tyP1026McSetTeach.tyMotionStdTrav.tyBtnJogFront.uiMaskRtStat));
	END_IF

	// Interlock When Moving
	IF tyP1026McSetTeach.tyMotionStdTrav.tyBtnOrigin.bRtCompl = TRUE THEN
		fUIInRtStatOff(ADR(tyP1026McSetTeach.tyMotionStdTrav.tyBtnMovAbs.uiMaskRtStat));
		fUIInRtStatOff(ADR(tyP1026McSetTeach.tyMotionStdTrav.tyBtnMovRel.uiMaskRtStat));
		fUIInRtStatOff(ADR(tyP1026McSetTeach.tyMotionStdTrav.tyBtnJogFront.uiMaskRtStat));
		fUIInRtStatOff(ADR(tyP1026McSetTeach.tyMotionStdTrav.tyBtnJogRear.uiMaskRtStat));
		fUIInRtStatOff(ADR(tyP1026McSetTeach.tyTeachTravPosA.tyBtn2.uiMaskRtStat));
		fUIInRtStatOff(ADR(tyP1026McSetTeach.tyTeachTravPosB.tyBtn2.uiMaskRtStat));

	ELSIF tyP1026McSetTeach.tyMotionStdTrav.tyBtnMovAbs.bRtCompl = TRUE THEN
		fUIInRtStatOff(ADR(tyP1026McSetTeach.tyMotionStdTrav.tyBtnOrigin.uiMaskRtStat));
		fUIInRtStatOff(ADR(tyP1026McSetTeach.tyMotionStdTrav.tyBtnMovRel.uiMaskRtStat));
		fUIInRtStatOff(ADR(tyP1026McSetTeach.tyMotionStdTrav.tyBtnJogFront.uiMaskRtStat));
		fUIInRtStatOff(ADR(tyP1026McSetTeach.tyMotionStdTrav.tyBtnJogRear.uiMaskRtStat));
		fUIInRtStatOff(ADR(tyP1026McSetTeach.tyTeachTravPosA.tyBtn2.uiMaskRtStat));
		fUIInRtStatOff(ADR(tyP1026McSetTeach.tyTeachTravPosB.tyBtn2.uiMaskRtStat));

	ELSIF tyP1026McSetTeach.tyMotionStdTrav.tyBtnMovRel.bRtCompl = TRUE THEN
		fUIInRtStatOff(ADR(tyP1026McSetTeach.tyMotionStdTrav.tyBtnOrigin.uiMaskRtStat));
		fUIInRtStatOff(ADR(tyP1026McSetTeach.tyMotionStdTrav.tyBtnMovAbs.uiMaskRtStat));
		fUIInRtStatOff(ADR(tyP1026McSetTeach.tyMotionStdTrav.tyBtnJogFront.uiMaskRtStat));
		fUIInRtStatOff(ADR(tyP1026McSetTeach.tyMotionStdTrav.tyBtnJogRear.uiMaskRtStat));
		fUIInRtStatOff(ADR(tyP1026McSetTeach.tyTeachTravPosA.tyBtn2.uiMaskRtStat));
		fUIInRtStatOff(ADR(tyP1026McSetTeach.tyTeachTravPosB.tyBtn2.uiMaskRtStat));

	ELSIF tyP1026McSetTeach.tyMotionStdTrav.tyBtnJogRear.bRtCompl = TRUE OR tyP1026McSetTeach.tyMotionStdTrav.tyBtnJogRear.bValue = TRUE THEN
		fUIInRtStatOff(ADR(tyP1026McSetTeach.tyMotionStdTrav.tyBtnOrigin.uiMaskRtStat));
		fUIInRtStatOff(ADR(tyP1026McSetTeach.tyMotionStdTrav.tyBtnMovAbs.uiMaskRtStat));
		fUIInRtStatOff(ADR(tyP1026McSetTeach.tyMotionStdTrav.tyBtnMovRel.uiMaskRtStat));
		fUIInRtStatOff(ADR(tyP1026McSetTeach.tyMotionStdTrav.tyBtnJogFront.uiMaskRtStat));
		fUIInRtStatOff(ADR(tyP1026McSetTeach.tyTeachTravPosA.tyBtn2.uiMaskRtStat));
		fUIInRtStatOff(ADR(tyP1026McSetTeach.tyTeachTravPosB.tyBtn2.uiMaskRtStat));

	ELSIF tyP1026McSetTeach.tyMotionStdTrav.tyBtnJogFront.bRtCompl = TRUE OR tyP1026McSetTeach.tyMotionStdTrav.tyBtnJogFront.bValue = TRUE THEN
		fUIInRtStatOff(ADR(tyP1026McSetTeach.tyMotionStdTrav.tyBtnOrigin.uiMaskRtStat));
		fUIInRtStatOff(ADR(tyP1026McSetTeach.tyMotionStdTrav.tyBtnMovAbs.uiMaskRtStat));
		fUIInRtStatOff(ADR(tyP1026McSetTeach.tyMotionStdTrav.tyBtnMovRel.uiMaskRtStat));
		fUIInRtStatOff(ADR(tyP1026McSetTeach.tyMotionStdTrav.tyBtnJogRear.uiMaskRtStat));
		fUIInRtStatOff(ADR(tyP1026McSetTeach.tyTeachTravPosA.tyBtn2.uiMaskRtStat));
		fUIInRtStatOff(ADR(tyP1026McSetTeach.tyTeachTravPosB.tyBtn2.uiMaskRtStat));

	ELSIF tyP1026McSetTeach.tyTeachTravPosA.tyBtn2.bRtCompl = TRUE THEN
		fUIInRtStatOff(ADR(tyP1026McSetTeach.tyMotionStdTrav.tyBtnOrigin.uiMaskRtStat));
		fUIInRtStatOff(ADR(tyP1026McSetTeach.tyMotionStdTrav.tyBtnMovAbs.uiMaskRtStat));
		fUIInRtStatOff(ADR(tyP1026McSetTeach.tyMotionStdTrav.tyBtnMovRel.uiMaskRtStat));
		fUIInRtStatOff(ADR(tyP1026McSetTeach.tyMotionStdTrav.tyBtnJogFront.uiMaskRtStat));
		fUIInRtStatOff(ADR(tyP1026McSetTeach.tyMotionStdTrav.tyBtnJogRear.uiMaskRtStat));

	ELSIF tyP1026McSetTeach.tyTeachTravPosB.tyBtn2.bRtCompl = TRUE THEN
		fUIInRtStatOff(ADR(tyP1026McSetTeach.tyMotionStdTrav.tyBtnOrigin.uiMaskRtStat));
		fUIInRtStatOff(ADR(tyP1026McSetTeach.tyMotionStdTrav.tyBtnMovAbs.uiMaskRtStat));
		fUIInRtStatOff(ADR(tyP1026McSetTeach.tyMotionStdTrav.tyBtnMovRel.uiMaskRtStat));
		fUIInRtStatOff(ADR(tyP1026McSetTeach.tyMotionStdTrav.tyBtnJogFront.uiMaskRtStat));
		fUIInRtStatOff(ADR(tyP1026McSetTeach.tyMotionStdTrav.tyBtnJogRear.uiMaskRtStat));

	END_IF

	//Axis Error
	IF tyP1026McSetTeach.tyMotionStdTrav.tyBtnPwr.bRtCompl = TRUE  THEN
		fUIInRtStatOff(ADR(tyP1026McSetTeach.tyMotionStdTrav.tyBtnRst.uiMaskRtStat));
	ELSE
		fUIInRtStatHide(ADR(tyP1026McSetTeach.tyMotionStdTrav.tyBtnRst.uiMaskRtStat));
	END_IF

	//Interlock Button Get
	IF p_bTravAxisErr = TRUE OR p_bTravIsHomed = FALSE OR p_bTravFwdLmtSen = TRUE OR p_bTravRevLmtSen = TRUE THEN
		fUIInRtStatOff(ADR(tyP1026McSetTeach.tyTeachTravPosA.tyBtn1.uiMaskRtStat));
		fUIInRtStatOff(ADR(tyP1026McSetTeach.tyTeachTravPosB.tyBtn1.uiMaskRtStat));
	ELSE
		fUIInRtStatHide(ADR(tyP1026McSetTeach.tyTeachTravPosA.tyBtn1.uiMaskRtStat));
		fUIInRtStatHide(ADR(tyP1026McSetTeach.tyTeachTravPosB.tyBtn1.uiMaskRtStat));
	END_IF

END_ACTION
```

#### Act_OptP1026TravUpdtDat.st
```iecst
ACTION Act_OptP1026TravUpdtDat:

	tyP1026McSetTeach.tyMotionStdTrav.tyNumCurrPos.diValue			:= p_diTravActualPos;
	tyP1026McSetTeach.tyMotionStdTrav.tyNumErrCode.diValue			:= UDINT_TO_DINT(p_udiTravAxisErrID);
	tyP1026McSetTeach.tyMotionStdTrav.tyBitmapPwr.usiValueIdx		:= BOOL_TO_USINT(p_bTravPwrOn);
	tyP1026McSetTeach.tyMotionStdTrav.tyBitmapRst.usiValueIdx		:= BOOL_TO_USINT(NOT p_bTravAxisErr);
	tyP1026McSetTeach.tyMotionStdTrav.tyBitmapOrigin.usiValueIdx	:= BOOL_TO_USINT(p_bTravIsHomed);
	tyP1026McSetTeach.tyMotionStdTrav.tyBtnFrontLmtSen.bValue		:= p_bTravFrontSen;
	tyP1026McSetTeach.tyMotionStdTrav.tyBtnRearLmtSen.bValue		:= p_bTravRearSen;

	//Machine Bitmap
	IF p_bTravIsHomed = TRUE THEN
		IF p_diTravActualPos <= (p_tyNtParamCurr.tyUITravTargetPos.diMax / 3) THEN
			tyP1026McSetTeach.tyMotionStdTrav.tyBitmapMc.uiValueIdx 	:= 5;
		ELSIF p_diTravActualPos <= (p_tyNtParamCurr.tyUITravTargetPos.diMax / 3 * 2) THEN
			tyP1026McSetTeach.tyMotionStdTrav.tyBitmapMc.uiValueIdx 	:= 6;
		ELSE
			tyP1026McSetTeach.tyMotionStdTrav.tyBitmapMc.uiValueIdx 	:= 7;
		END_IF
	ELSE
		tyP1026McSetTeach.tyMotionStdTrav.tyBitmapMc.uiValueIdx	:= 5;
	END_IF

	IF p_tyNtParamCurr.eProjMag = ULMagDual THEN
		IF p_tyNtParamCurr.bProjLifterMagPlatform AND p_tyNtParamCurr.bUIConvDirRL THEN
			IF 	tyP1026McSetTeach.tyMotionStdTrav.tyBitmapMc.uiValueIdx < 700 THEN
				tyP1026McSetTeach.tyMotionStdTrav.tyBitmapMc.uiValueIdx	:= tyP1026McSetTeach.tyMotionStdTrav.tyBitmapMc.uiValueIdx + 700;
			END_IF
		ELSIF p_tyNtParamCurr.bProjLifterMagPlatform THEN
			IF 	tyP1026McSetTeach.tyMotionStdTrav.tyBitmapMc.uiValueIdx < 600 THEN
				tyP1026McSetTeach.tyMotionStdTrav.tyBitmapMc.uiValueIdx	:= tyP1026McSetTeach.tyMotionStdTrav.tyBitmapMc.uiValueIdx + 600;
			END_IF
		ELSIF p_tyNtParamCurr.bMagAutoVerifyPrep = FALSE THEN
			IF 	tyP1026McSetTeach.tyMotionStdTrav.tyBitmapMc.uiValueIdx < 100 THEN
				tyP1026McSetTeach.tyMotionStdTrav.tyBitmapMc.uiValueIdx	:= tyP1026McSetTeach.tyMotionStdTrav.tyBitmapMc.uiValueIdx + 300;
			END_IF
		ELSE
			IF 	tyP1026McSetTeach.tyMotionStdTrav.tyBitmapMc.uiValueIdx < 300 THEN
				tyP1026McSetTeach.tyMotionStdTrav.tyBitmapMc.uiValueIdx	:= tyP1026McSetTeach.tyMotionStdTrav.tyBitmapMc.uiValueIdx + 300;
			END_IF
		END_IF
	ELSIF p_tyNtParamCurr.eProjMag = ULMagTriple THEN
		IF p_tyNtParamCurr.bProjLifterMagPlatform AND p_tyNtParamCurr.bUIConvDirRL THEN
			IF 	tyP1026McSetTeach.tyMotionStdTrav.tyBitmapMc.uiValueIdx < 800 THEN
				tyP1026McSetTeach.tyMotionStdTrav.tyBitmapMc.uiValueIdx	:= tyP1026McSetTeach.tyMotionStdTrav.tyBitmapMc.uiValueIdx + 800;
			END_IF
		ELSIF p_tyNtParamCurr.bProjLifterMagPlatform THEN
			IF 	tyP1026McSetTeach.tyMotionStdTrav.tyBitmapMc.uiValueIdx < 500 THEN
				tyP1026McSetTeach.tyMotionStdTrav.tyBitmapMc.uiValueIdx	:= tyP1026McSetTeach.tyMotionStdTrav.tyBitmapMc.uiValueIdx + 500;
			END_IF
		ELSIF p_tyNtParamCurr.bMagAutoVerifyPrep = TRUE AND p_tyNtParamCurr.bProjMotorizedPusherPrep = FALSE THEN
			IF 	tyP1026McSetTeach.tyMotionStdTrav.tyBitmapMc.uiValueIdx < 200 THEN
				tyP1026McSetTeach.tyMotionStdTrav.tyBitmapMc.uiValueIdx	:= tyP1026McSetTeach.tyMotionStdTrav.tyBitmapMc.uiValueIdx + 200;
			END_IF
		ELSIF p_tyNtParamCurr.bMagAutoVerifyPrep = FALSE AND p_tyNtParamCurr.bProjMotorizedPusherPrep = TRUE THEN
			IF 	tyP1026McSetTeach.tyMotionStdTrav.tyBitmapMc.uiValueIdx < 400 THEN
				tyP1026McSetTeach.tyMotionStdTrav.tyBitmapMc.uiValueIdx	:= tyP1026McSetTeach.tyMotionStdTrav.tyBitmapMc.uiValueIdx + 400;
			END_IF
		END_IF
	END_IF

END_ACTION
```

#### Act_OptP1026TravKeypad.st
```iecst
ACTION Act_OptP1026TravKeypad:

	IF fUIOutRtStatTPIsOpen(ADR(tyP1026McSetTeach.tyMotionStdTrav.tyNumTargetPos.uiRtStat)) = TRUE THEN
		tyProperty.tyKeypad.tyStringTitle.sKeypadTitle		:= tyP1026McSetTeach.tyMotionStdTrav.tyNumTargetPos.sKeypadTitle;

	ELSIF fUIOutRtStatTPIsOpen(ADR(tyP1026McSetTeach.tyMotionStdTrav.tyNumStepSize.uiRtStat)) = TRUE THEN
		tyProperty.tyKeypad.tyStringTitle.sKeypadTitle		:= tyP1026McSetTeach.tyMotionStdTrav.tyNumStepSize.sKeypadTitle;

	ELSIF fUIOutRtStatTPIsOpen(ADR(tyP1026McSetTeach.tyMotionStdTrav.tyNumNomSpd.uiRtStat)) = TRUE THEN
		tyProperty.tyKeypad.tyStringTitle.sKeypadTitle		:= tyP1026McSetTeach.tyMotionStdTrav.tyNumNomSpd.sKeypadTitle;

	ELSIF fUIOutRtStatTPIsOpen(ADR(tyP1026McSetTeach.tyMotionStdTrav.tyNumSlwSpd.uiRtStat)) = TRUE THEN
		tyProperty.tyKeypad.tyStringTitle.sKeypadTitle		:= tyP1026McSetTeach.tyMotionStdTrav.tyNumSlwSpd.sKeypadTitle;

	END_IF

END_ACTION
```

#### Act_OptP1026TravRstMnl.st
```iecst
ACTION Act_OptP1026TravRstMnl:

	IF EDGEPOS((bManualMod = FALSE) OR (p_eTravStatus = Error)) THEN

		bJogSlow				:= FALSE;
		bJogFast				:= FALSE;
		fbJogSlowToFastDlyTm.IN	:= FALSE;

		tyP1026McSetTeach.tyMotionStdTrav.tyBtnPwr.bRtCompl				:= FALSE;
		tyP1026McSetTeach.tyMotionStdTrav.tyBtnStop.bRtCompl			:= FALSE;
		tyP1026McSetTeach.tyMotionStdTrav.tyBtnOrigin.bRtCompl			:= FALSE;
		tyP1026McSetTeach.tyMotionStdTrav.tyBtnRst.bRtCompl				:= FALSE;
		tyP1026McSetTeach.tyMotionStdTrav.tyBtnMovAbs.bRtCompl			:= FALSE;
		tyP1026McSetTeach.tyMotionStdTrav.tyBtnMovRel.bRtCompl			:= FALSE;
		tyP1026McSetTeach.tyMotionStdTrav.tyBtnJogFront.bRtCompl		:= FALSE;
		tyP1026McSetTeach.tyMotionStdTrav.tyBtnJogRear.bRtCompl			:= FALSE;

		tyP1026McSetTeach.tyTeachTravPosA.tyBtn2.bRtCompl				:= FALSE;
		tyP1026McSetTeach.tyTeachTravPosB.tyBtn2.bRtCompl				:= FALSE;

		tyP1026McSetTeach.tyMotionStdTrav.tyBtnPwr.bValue				:= FALSE;
		tyP1026McSetTeach.tyMotionStdTrav.tyBtnStop.bValue				:= TRUE;
		tyP1026McSetTeach.tyMotionStdTrav.tyBtnOrigin.bValue			:= FALSE;
		tyP1026McSetTeach.tyMotionStdTrav.tyBtnRst.bValue				:= FALSE;
		tyP1026McSetTeach.tyMotionStdTrav.tyBtnMovAbs.bValue			:= FALSE;
		tyP1026McSetTeach.tyMotionStdTrav.tyBtnMovRel.bValue			:= FALSE;
		tyP1026McSetTeach.tyMotionStdTrav.tyBtnJogFront.bValue			:= FALSE;
		tyP1026McSetTeach.tyMotionStdTrav.tyBtnJogRear.bValue			:= FALSE;

		tyP1026McSetTeach.tyTeachTravPosA.tyBtn2.bValue					:= FALSE;
		tyP1026McSetTeach.tyTeachTravPosB.tyBtn2.bValue					:= FALSE;

		tyP1026McSetTeach.tyMotionStdTrav.tyBtnPwr.bRtLk				:= FALSE;
		tyP1026McSetTeach.tyMotionStdTrav.tyBtnStop.bRtLk				:= TRUE;
		tyP1026McSetTeach.tyMotionStdTrav.tyBtnOrigin.bRtLk				:= FALSE;
		tyP1026McSetTeach.tyMotionStdTrav.tyBtnRst.bRtLk				:= FALSE;
		tyP1026McSetTeach.tyMotionStdTrav.tyBtnMovAbs.bRtLk				:= FALSE;
		tyP1026McSetTeach.tyMotionStdTrav.tyBtnMovRel.bRtLk				:= FALSE;
		tyP1026McSetTeach.tyMotionStdTrav.tyBtnJogFront.bRtLk			:= FALSE;
		tyP1026McSetTeach.tyMotionStdTrav.tyBtnJogRear.bRtLk			:= FALSE;

		tyP1026McSetTeach.tyTeachTravPosA.tyBtn2.bRtLk					:= FALSE;
		tyP1026McSetTeach.tyTeachTravPosB.tyBtn2.bRtLk					:= FALSE;

		tyP1026McSetTeach.tyMotionStdTrav.tyBtnPwr.uiMaskRtStat			:= TRUE;
		tyP1026McSetTeach.tyMotionStdTrav.tyBtnOrigin.uiMaskRtStat		:= FALSE;
		tyP1026McSetTeach.tyMotionStdTrav.tyBtnRst.uiMaskRtStat			:= TRUE;
		tyP1026McSetTeach.tyMotionStdTrav.tyBtnMovAbs.uiMaskRtStat		:= FALSE;
		tyP1026McSetTeach.tyMotionStdTrav.tyBtnMovRel.uiMaskRtStat		:= FALSE;
		tyP1026McSetTeach.tyMotionStdTrav.tyBtnJogFront.uiMaskRtStat	:= FALSE;
		tyP1026McSetTeach.tyMotionStdTrav.tyBtnJogRear.uiMaskRtStat		:= FALSE;

		tyP1026McSetTeach.tyTeachTravPosA.tyBtn2.uiMaskRtStat			:= FALSE;
		tyP1026McSetTeach.tyTeachTravPosB.tyBtn2.uiMaskRtStat			:= FALSE;

	END_IF

END_ACTION
```

#### Act_OptP1026LifterTeach.st
```iecst
ACTION Act_OptP1026LifterTeach:

	IF tyP1026McSetTeach.tyTeachLifterPosA.tyBtn1.bRtCompl = TRUE THEN

		p_tyC0008MsgBox ACCESS ADR(tyP1026McSetTeach.tyMsgBoxUpdtLifterPosA);
		IF tyP1026McSetTeach.tyMsgBoxUpdtLifterPosA.tyBtnNo.bRtCompl THEN	//tyBtnNo
			tyP1026McSetTeach.tyMsgBoxUpdtLifterPosA.tyBtnNo.bRtCompl	:= FALSE;
			tyP1026McSetTeach.tyMsgBoxUpdtLifterPosA.tyBtnNo.bValue		:= FALSE;

			p_tyC0008MsgBox ACCESS ADR(tyP1026McSetTeach.tyMsgBoxHide);

			//Write Actual Position To Machine Settings
			tyP1021McSetGen.tyGen.tyNumLiftPosLaneA.diValue		:= p_diLifterBtmActualPos;
			tyP1021McSetGen.tyGen.tyNumLiftPosLaneA.bRtCompl	:= TRUE;

			//Back To Machine Settings
			eChgPage	:= UIP1021McSetGen;

			fUIInRtStatHide(ADR(tyCommon.tySet.tyBtnSave.uiMaskRtStat));

			tyP1026McSetTeach.tyTeachLifterPosA.tyBtn1.bRtCompl	:= FALSE;
			tyP1026McSetTeach.tyTeachLifterPosA.tyBtn1.bValue	:= FALSE;
//		ELSIF tyP1026McSetTeach.tyMsgBoxUpdtLifterPosA.tyBtnNo.bRtCompl THEN
//			tyP1026McSetTeach.tyMsgBoxUpdtLifterPosA.tyBtnNo.bRtCompl	:= FALSE;
//			tyP1026McSetTeach.tyMsgBoxUpdtLifterPosA.tyBtnNo.bValue		:= FALSE;
//
//			p_tyC0008MsgBox ACCESS ADR(tyP1026McSetTeach.tyMsgBoxHide);
//
//			//Back To Machine Settings
//			eChgPage	:= UIP1021McSetGen;
//
//			tyP1026McSetTeach.tyTeachLifterPosA.tyBtn1.bRtCompl	:= FALSE;
//			tyP1026McSetTeach.tyTeachLifterPosA.tyBtn1.bValue	:= FALSE;

		END_IF

	ELSIF tyP1026McSetTeach.tyTeachLifterPosB.tyBtn1.bRtCompl = TRUE THEN

		p_tyC0008MsgBox ACCESS ADR(tyP1026McSetTeach.tyMsgBoxUpdtLifterPosB);
		IF tyP1026McSetTeach.tyMsgBoxUpdtLifterPosB.tyBtnNo.bRtCompl THEN
			tyP1026McSetTeach.tyMsgBoxUpdtLifterPosB.tyBtnNo.bRtCompl	:= FALSE;
			tyP1026McSetTeach.tyMsgBoxUpdtLifterPosB.tyBtnNo.bValue		:= FALSE;

			p_tyC0008MsgBox ACCESS ADR(tyP1026McSetTeach.tyMsgBoxHide);

			//Write Actual Position To Machine Settings
			tyP1021McSetGen.tyGen.tyNumLiftPosLaneB.diValue		:= p_diLifterBtmActualPos;
			tyP1021McSetGen.tyGen.tyNumLiftPosLaneB.bRtCompl	:= TRUE;

			//Back To Machine Settings
			eChgPage	:= UIP1021McSetGen;

			fUIInRtStatHide(ADR(tyCommon.tySet.tyBtnSave.uiMaskRtStat));

			tyP1026McSetTeach.tyTeachLifterPosB.tyBtn1.bRtCompl	:= FALSE;
			tyP1026McSetTeach.tyTeachLifterPosB.tyBtn1.bValue	:= FALSE;

//		ELSIF tyP1026McSetTeach.tyMsgBoxUpdtLifterPosB.tyBtnNo.bRtCompl THEN
//			tyP1026McSetTeach.tyMsgBoxUpdtLifterPosB.tyBtnNo.bRtCompl	:= FALSE;
//			tyP1026McSetTeach.tyMsgBoxUpdtLifterPosB.tyBtnNo.bValue		:= FALSE;
//
//			p_tyC0008MsgBox ACCESS ADR(tyP1026McSetTeach.tyMsgBoxHide);
//
//			//Back To Machine Settings
//			eChgPage	:= UIP1021McSetGen;
//
//			tyP1026McSetTeach.tyTeachLifterPosB.tyBtn1.bRtCompl	:= FALSE;
//			tyP1026McSetTeach.tyTeachLifterPosB.tyBtn1.bValue	:= FALSE;

		END_IF

	ELSIF tyP1026McSetTeach.tyTeachLifterTopPos.tyBtn1.bRtCompl = TRUE THEN

		p_tyC0008MsgBox ACCESS ADR(tyP1026McSetTeach.tyMsgBoxUpdtLifterTopPos);
		IF tyP1026McSetTeach.tyMsgBoxUpdtLifterTopPos.tyBtnNo.bRtCompl THEN
			tyP1026McSetTeach.tyMsgBoxUpdtLifterTopPos.tyBtnNo.bRtCompl		:= FALSE;
			tyP1026McSetTeach.tyMsgBoxUpdtLifterTopPos.tyBtnNo.bValue		:= FALSE;

			p_tyC0008MsgBox ACCESS ADR(tyP1026McSetTeach.tyMsgBoxHide);

			//Write Actual Position To Machine Settings
			tyP1021McSetGen.tyGen.tyNumLifterTopPos.diValue		:= p_diLifterBtmActualPos;
			tyP1021McSetGen.tyGen.tyNumLifterTopPos.bRtCompl	:= TRUE;

			//Back To Machine Settings
			eChgPage	:= UIP1021McSetGen;

			fUIInRtStatHide(ADR(tyCommon.tySet.tyBtnSave.uiMaskRtStat));

			tyP1026McSetTeach.tyTeachLifterTopPos.tyBtn1.bRtCompl	:= FALSE;
			tyP1026McSetTeach.tyTeachLifterTopPos.tyBtn1.bValue	:= FALSE;

//		ELSIF tyP1026McSetTeach.tyMsgBoxUpdtLifterTopPos.tyBtnNo.bRtCompl THEN
//			tyP1026McSetTeach.tyMsgBoxUpdtLifterTopPos.tyBtnNo.bRtCompl		:= FALSE;
//			tyP1026McSetTeach.tyMsgBoxUpdtLifterTopPos.tyBtnNo.bValue		:= FALSE;
//
//			p_tyC0008MsgBox ACCESS ADR(tyP1026McSetTeach.tyMsgBoxHide);
//
//			//Back To Machine Settings
//			eChgPage	:= UIP1021McSetGen;
//
//			tyP1026McSetTeach.tyTeachLifterTopPos.tyBtn1.bRtCompl	:= FALSE;
//			tyP1026McSetTeach.tyTeachLifterTopPos.tyBtn1.bValue	:= FALSE;

		END_IF

	ELSIF tyP1026McSetTeach.tyTeachLifterBtmPos.tyBtn1.bRtCompl = TRUE THEN

		p_tyC0008MsgBox ACCESS ADR(tyP1026McSetTeach.tyMsgBoxUpdtLifterBtmPos);
		IF tyP1026McSetTeach.tyMsgBoxUpdtLifterBtmPos.tyBtnNo.bRtCompl THEN
			tyP1026McSetTeach.tyMsgBoxUpdtLifterBtmPos.tyBtnNo.bRtCompl		:= FALSE;
			tyP1026McSetTeach.tyMsgBoxUpdtLifterBtmPos.tyBtnNo.bValue		:= FALSE;

			p_tyC0008MsgBox ACCESS ADR(tyP1026McSetTeach.tyMsgBoxHide);

			//Write Actual Position To Machine Settings
			tyP1021McSetGen.tyGen.tyNumLifterBtmPos.diValue		:= p_diLifterBtmActualPos;
			tyP1021McSetGen.tyGen.tyNumLifterBtmPos.bRtCompl	:= TRUE;

			//Back To Machine Settings
			eChgPage	:= UIP1021McSetGen;

			fUIInRtStatHide(ADR(tyCommon.tySet.tyBtnSave.uiMaskRtStat));

			tyP1026McSetTeach.tyTeachLifterBtmPos.tyBtn1.bRtCompl	:= FALSE;
			tyP1026McSetTeach.tyTeachLifterBtmPos.tyBtn1.bValue	:= FALSE;

//		ELSIF tyP1026McSetTeach.tyMsgBoxUpdtLifterBtmPos.tyBtnNo.bRtCompl THEN
//			tyP1026McSetTeach.tyMsgBoxUpdtLifterBtmPos.tyBtnNo.bRtCompl		:= FALSE;
//			tyP1026McSetTeach.tyMsgBoxUpdtLifterBtmPos.tyBtnNo.bValue		:= FALSE;
//
//			p_tyC0008MsgBox ACCESS ADR(tyP1026McSetTeach.tyMsgBoxHide);
//
//			//Write Actual Position To Machine Settings
//			tyP1021McSetGen.tyGen.tyNumLifterBtmPos.diValue		:= p_diLifterBtmActualPos;
//			tyP1021McSetGen.tyGen.tyNumLifterBtmPos.bRtCompl	:= TRUE;
//
//			//Back To Machine Settings
//			eChgPage	:= UIP1021McSetGen;
//
//			fUIInRtStatHide(ADR(tyCommon.tySet.tyBtnSave.uiMaskRtStat));
//
//			tyP1026McSetTeach.tyTeachLifterBtmPos.tyBtn1.bRtCompl	:= FALSE;
//			tyP1026McSetTeach.tyTeachLifterBtmPos.tyBtn1.bValue	:= FALSE;

		END_IF

	ELSIF tyP1026McSetTeach.tyTeachLifterTopPos2.tyBtn1.bRtCompl = TRUE THEN

		p_tyC0008MsgBox ACCESS ADR(tyP1026McSetTeach.tyMsgBoxUpdtLifterTopPos2);
		IF tyP1026McSetTeach.tyMsgBoxUpdtLifterTopPos2.tyBtnNo.bRtCompl THEN
			tyP1026McSetTeach.tyMsgBoxUpdtLifterTopPos2.tyBtnNo.bRtCompl		:= FALSE;
			tyP1026McSetTeach.tyMsgBoxUpdtLifterTopPos2.tyBtnNo.bValue		:= FALSE;

			p_tyC0008MsgBox ACCESS ADR(tyP1026McSetTeach.tyMsgBoxHide);

			//Write Actual Position To Machine Settings
			tyP1021McSetGen.tyGen.tyNumLifterTopPos2.diValue		:= p_diLifter2ActualPos;
			tyP1021McSetGen.tyGen.tyNumLifterTopPos2.bRtCompl	:= TRUE;

			//Back To Machine Settings
			eChgPage	:= UIP1021McSetGen;

			fUIInRtStatHide(ADR(tyCommon.tySet.tyBtnSave.uiMaskRtStat));

			tyP1026McSetTeach.tyTeachLifterTopPos2.tyBtn1.bRtCompl	:= FALSE;
			tyP1026McSetTeach.tyTeachLifterTopPos2.tyBtn1.bValue	:= FALSE;
//		ELSIF tyP1026McSetTeach.tyMsgBoxUpdtLifterTopPos2.tyBtnNo.bRtCompl THEN
//			tyP1026McSetTeach.tyMsgBoxUpdtLifterTopPos2.tyBtnNo.bRtCompl		:= FALSE;
//			tyP1026McSetTeach.tyMsgBoxUpdtLifterTopPos2.tyBtnNo.bValue		:= FALSE;
//
//			p_tyC0008MsgBox ACCESS ADR(tyP1026McSetTeach.tyMsgBoxHide);
//
//			//Back To Machine Settings
//			eChgPage	:= UIP1021McSetGen;
//
//			tyP1026McSetTeach.tyTeachLifterTopPos2.tyBtn1.bRtCompl	:= FALSE;
//			tyP1026McSetTeach.tyTeachLifterTopPos2.tyBtn1.bValue	:= FALSE;
//
		END_IF

	ELSIF tyP1026McSetTeach.tyTeachLifterBtmPos2.tyBtn1.bRtCompl = TRUE THEN

		p_tyC0008MsgBox ACCESS ADR(tyP1026McSetTeach.tyMsgBoxUpdtLifterBtmPos2);
		IF tyP1026McSetTeach.tyMsgBoxUpdtLifterBtmPos2.tyBtnNo.bRtCompl THEN
			tyP1026McSetTeach.tyMsgBoxUpdtLifterBtmPos2.tyBtnNo.bRtCompl		:= FALSE;
			tyP1026McSetTeach.tyMsgBoxUpdtLifterBtmPos2.tyBtnNo.bValue		:= FALSE;

			p_tyC0008MsgBox ACCESS ADR(tyP1026McSetTeach.tyMsgBoxHide);

			//Write Actual Position To Machine Settings
			tyP1021McSetGen.tyGen.tyNumLifterBtmPos2.diValue		:= p_diLifter2ActualPos;
			tyP1021McSetGen.tyGen.tyNumLifterBtmPos2.bRtCompl	:= TRUE;

			//Back To Machine Settings
			eChgPage	:= UIP1021McSetGen;

			fUIInRtStatHide(ADR(tyCommon.tySet.tyBtnSave.uiMaskRtStat));

			tyP1026McSetTeach.tyTeachLifterBtmPos2.tyBtn1.bRtCompl	:= FALSE;
			tyP1026McSetTeach.tyTeachLifterBtmPos2.tyBtn1.bValue	:= FALSE;
//		ELSIF tyP1026McSetTeach.tyMsgBoxUpdtLifterBtmPos2.tyBtnNo.bRtCompl THEN
//			tyP1026McSetTeach.tyMsgBoxUpdtLifterBtmPos2.tyBtnNo.bRtCompl		:= FALSE;
//			tyP1026McSetTeach.tyMsgBoxUpdtLifterBtmPos2.tyBtnNo.bValue		:= FALSE;
//
//			p_tyC0008MsgBox ACCESS ADR(tyP1026McSetTeach.tyMsgBoxHide);
//
//			//Back To Machine Settings
//			eChgPage	:= UIP1021McSetGen;
//
//			tyP1026McSetTeach.tyTeachLifterBtmPos2.tyBtn1.bRtCompl	:= FALSE;
//			tyP1026McSetTeach.tyTeachLifterBtmPos2.tyBtn1.bValue	:= FALSE;
//
		END_IF
	END_IF

END_ACTION
```

#### Act_OptP1026LifterFBCtrl.st
```iecst
ACTION Act_OptP1026LifterFBCtrl:

	fbJogSlowToFastDlyTm.PT	:= T#2s;
	fbJogSlowToFastDlyTm;
	fbLmtRstTm;

	//Lifter Safety Sensor Interruption
	IF EDGENEG(p_tyDI.bLifterSafetyLmtSW1 AND p_tyDI.bLifterSafetyLmtSW2 AND p_tyDI.bLifterTimingBeltSen) THEN
		tyP1026McSetTeach.tyMotionStdLifter.tyBtnStop.bRtCompl	:= TRUE;
	END_IF

	IF EDGEPOS((p_udiLifterBtmAxisErrID = 21570 OR p_udiLifterBtmAxisErrID = 21571) AND tyP1026McSetTeach.tyMotionStdLifter.tyBtnJogDown.bValue = FALSE AND tyP1026McSetTeach.tyMotionStdLifter.tyBtnJogUp.bValue = FALSE) THEN
		fbLmtRstTm.IN	:= TRUE;
	END_IF

	IF fbLmtRstTm.Q = TRUE THEN
		tyP1026McSetTeach.tyMotionStdLifter.tyBtnRst.bRtCompl	:= TRUE;
	END_IF

	IF (tyP1026McSetTeach.tyMotionStdLifter.tyBtnJogUp.bValue = FALSE AND tyP1026McSetTeach.tyMotionStdLifter.tyBtnJogDown.bValue = FALSE) AND (p_bLifterBtmJogging = TRUE) THEN
		bJogStopLifter	:= TRUE;
	END_IF

	IF tyP1026McSetTeach.tyMotionStdLifter.tyBtnStop.bRtCompl = TRUE THEN
		eLifterBtmAct		:= LifterActStop;

		IF p_eLifterBtmStat = LifterActStop AND p_eLifterBtmStatus = Done THEN
			eLifterBtmAct	:= LifterActIdle;

			tyP1026McSetTeach.tyMotionStdLifter.tyBtnStop.bRtCompl			:= FALSE;
			tyP1026McSetTeach.tyMotionStdLifter.tyBtnJogDown.bRtCompl		:= FALSE;
			tyP1026McSetTeach.tyMotionStdLifter.tyBtnJogUp.bRtCompl			:= FALSE;
			tyP1026McSetTeach.tyMotionStdLifter.tyBtnOrigin.bRtCompl		:= FALSE;
			tyP1026McSetTeach.tyMotionStdLifter.tyBtnMovAbs.bRtCompl		:= FALSE;
			tyP1026McSetTeach.tyMotionStdLifter.tyBtnMovRel.bRtCompl		:= FALSE;

			tyP1026McSetTeach.tyTeachLifterPosA.tyBtn2.bRtCompl				:= FALSE;
			tyP1026McSetTeach.tyTeachLifterPosB.tyBtn2.bRtCompl				:= FALSE;
			tyP1026McSetTeach.tyTeachLifterTopPos.tyBtn2.bRtCompl				:= FALSE;//
			tyP1026McSetTeach.tyTeachLifterBtmPos.tyBtn2.bRtCompl				:= FALSE;//

			tyP1026McSetTeach.tyMotionStdLifter.tyBtnStop.bValue			:= TRUE;
			tyP1026McSetTeach.tyMotionStdLifter.tyBtnJogDown.bValue			:= FALSE;
			tyP1026McSetTeach.tyMotionStdLifter.tyBtnJogUp.bValue			:= FALSE;
			tyP1026McSetTeach.tyMotionStdLifter.tyBtnOrigin.bValue			:= FALSE;
			tyP1026McSetTeach.tyMotionStdLifter.tyBtnMovAbs.bValue			:= FALSE;
			tyP1026McSetTeach.tyMotionStdLifter.tyBtnMovRel.bValue			:= FALSE;

			tyP1026McSetTeach.tyTeachLifterPosA.tyBtn2.bValue				:= FALSE;
			tyP1026McSetTeach.tyTeachLifterPosB.tyBtn2.bValue				:= FALSE;
			tyP1026McSetTeach.tyTeachLifterTopPos.tyBtn2.bValue				:= FALSE;
			tyP1026McSetTeach.tyTeachLifterBtmPos.tyBtn2.bValue				:= FALSE;

			tyP1026McSetTeach.tyMotionStdLifter.tyBtnStop.bRtLk				:= TRUE;
			tyP1026McSetTeach.tyMotionStdLifter.tyBtnJogDown.bRtLk			:= FALSE;
			tyP1026McSetTeach.tyMotionStdLifter.tyBtnJogUp.bRtLk			:= FALSE;
			tyP1026McSetTeach.tyMotionStdLifter.tyBtnOrigin.bRtLk			:= FALSE;
			tyP1026McSetTeach.tyMotionStdLifter.tyBtnMovAbs.bRtLk			:= FALSE;
			tyP1026McSetTeach.tyMotionStdLifter.tyBtnMovRel.bRtLk			:= FALSE;

			tyP1026McSetTeach.tyTeachLifterPosA.tyBtn2.bRtLk				:= FALSE;
			tyP1026McSetTeach.tyTeachLifterPosB.tyBtn2.bRtLk				:= FALSE;
			tyP1026McSetTeach.tyTeachLifterTopPos.tyBtn2.bRtLk				:= FALSE;
			tyP1026McSetTeach.tyTeachLifterBtmPos.tyBtn2.bRtLk				:= FALSE;

		END_IF

	ELSIF (tyP1026McSetTeach.tyMotionStdLifter.tyBtnJogDown.bRtCompl = TRUE) OR (tyP1026McSetTeach.tyMotionStdLifter.tyBtnJogUp.bRtCompl = TRUE) OR (bJogStopLifter = TRUE) THEN
		bJogSlow					:= FALSE;
		bJogFast					:= FALSE;
		fbJogSlowToFastDlyTm.IN		:= FALSE;

		eLifterBtmAct	:= LifterActJogStop;

		IF p_eLifterBtmStat = LifterActJogStop AND p_eLifterBtmStatus = Done THEN
			eLifterBtmAct		:= LifterActIdle;

			bJogStopLifter	:= FALSE;

			tyP1026McSetTeach.tyMotionStdLifter.tyBtnStop.bRtCompl			:= FALSE;
			tyP1026McSetTeach.tyMotionStdLifter.tyBtnJogDown.bRtCompl		:= FALSE;
			tyP1026McSetTeach.tyMotionStdLifter.tyBtnJogUp.bRtCompl			:= FALSE;
			tyP1026McSetTeach.tyMotionStdLifter.tyBtnOrigin.bRtCompl		:= FALSE;
			tyP1026McSetTeach.tyMotionStdLifter.tyBtnMovAbs.bRtCompl		:= FALSE;
			tyP1026McSetTeach.tyMotionStdLifter.tyBtnMovRel.bRtCompl		:= FALSE;

			tyP1026McSetTeach.tyTeachLifterPosA.tyBtn2.bRtCompl				:= FALSE;
			tyP1026McSetTeach.tyTeachLifterPosB.tyBtn2.bRtCompl				:= FALSE;
			tyP1026McSetTeach.tyTeachLifterTopPos.tyBtn2.bRtCompl				:= FALSE;//
			tyP1026McSetTeach.tyTeachLifterBtmPos.tyBtn2.bRtCompl				:= FALSE;//

			tyP1026McSetTeach.tyMotionStdLifter.tyBtnStop.bValue			:= TRUE;
			tyP1026McSetTeach.tyMotionStdLifter.tyBtnJogDown.bValue			:= FALSE;
			tyP1026McSetTeach.tyMotionStdLifter.tyBtnJogUp.bValue			:= FALSE;
			tyP1026McSetTeach.tyMotionStdLifter.tyBtnOrigin.bValue			:= FALSE;
			tyP1026McSetTeach.tyMotionStdLifter.tyBtnMovAbs.bValue			:= FALSE;
			tyP1026McSetTeach.tyMotionStdLifter.tyBtnMovRel.bValue			:= FALSE;

			tyP1026McSetTeach.tyTeachLifterPosA.tyBtn2.bValue				:= FALSE;
			tyP1026McSetTeach.tyTeachLifterPosB.tyBtn2.bValue				:= FALSE;
			tyP1026McSetTeach.tyTeachLifterTopPos.tyBtn2.bValue				:= FALSE;
			tyP1026McSetTeach.tyTeachLifterBtmPos.tyBtn2.bValue				:= FALSE;

			tyP1026McSetTeach.tyMotionStdLifter.tyBtnStop.bRtLk				:= TRUE;
			tyP1026McSetTeach.tyMotionStdLifter.tyBtnJogDown.bRtLk			:= FALSE;
			tyP1026McSetTeach.tyMotionStdLifter.tyBtnJogUp.bRtLk			:= FALSE;
			tyP1026McSetTeach.tyMotionStdLifter.tyBtnOrigin.bRtLk			:= FALSE;
			tyP1026McSetTeach.tyMotionStdLifter.tyBtnMovAbs.bRtLk			:= FALSE;
			tyP1026McSetTeach.tyMotionStdLifter.tyBtnMovRel.bRtLk			:= FALSE;

			tyP1026McSetTeach.tyTeachLifterPosA.tyBtn2.bRtLk				:= FALSE;
			tyP1026McSetTeach.tyTeachLifterPosB.tyBtn2.bRtLk				:= FALSE;
			tyP1026McSetTeach.tyTeachLifterTopPos.tyBtn2.bRtLk				:= FALSE;
			tyP1026McSetTeach.tyTeachLifterBtmPos.tyBtn2.bRtLk				:= FALSE;

		END_IF

	ELSIF tyP1026McSetTeach.tyMotionStdLifter.tyBtnPwr.bRtCompl = TRUE THEN
		tyP1026McSetTeach.tyMotionStdLifter.tyBtnPwr.bRtLk	:= TRUE;

		IF tyP1026McSetTeach.tyMotionStdLifter.tyBtnPwr.bValue = TRUE THEN
			eLifterBtmAct	:= LifterActPwrOn;

			IF p_eLifterBtmStat = LifterActPwrOn AND p_eLifterBtmStatus = Done THEN
				eLifterBtmAct	:= LifterActIdle;

				tyP1026McSetTeach.tyMotionStdLifter.tyBtnPwr.bRtCompl	:= FALSE;
				tyP1026McSetTeach.tyMotionStdLifter.tyBtnPwr.bRtLk		:= FALSE;
			END_IF
		ELSE
			eLifterBtmAct	:= LifterActPwrOff;

			IF p_eLifterBtmStat = LifterActPwrOff AND p_eLifterBtmStatus = Done THEN
				eLifterBtmAct	:= LifterActIdle;

				tyP1026McSetTeach.tyMotionStdLifter.tyBtnPwr.bRtCompl	:= FALSE;
				tyP1026McSetTeach.tyMotionStdLifter.tyBtnPwr.bRtLk		:= FALSE;
			END_IF
		END_IF

	ELSIF tyP1026McSetTeach.tyMotionStdLifter.tyBtnOrigin.bRtCompl = TRUE THEN
		tyP1026McSetTeach.tyMotionStdLifter.tyBtnOrigin.bValue	:= TRUE;
		tyP1026McSetTeach.tyMotionStdLifter.tyBtnStop.bValue	:= FALSE;

		tyP1026McSetTeach.tyMotionStdLifter.tyBtnOrigin.bRtLk	:= TRUE;
		tyP1026McSetTeach.tyMotionStdLifter.tyBtnStop.bRtLk		:= FALSE;

		eLifterBtmAct	:= LifterActHoming;

		IF p_eLifterBtmStat = LifterActHoming AND p_eLifterBtmStatus = Done THEN
			eLifterBtmAct	:= LifterActIdle;

			tyP1026McSetTeach.tyMotionStdLifter.tyBtnOrigin.bRtCompl	:= FALSE;
			tyP1026McSetTeach.tyMotionStdLifter.tyBtnOrigin.bValue		:= FALSE;
			tyP1026McSetTeach.tyMotionStdLifter.tyBtnStop.bValue		:= TRUE;

			tyP1026McSetTeach.tyMotionStdLifter.tyBtnOrigin.bRtLk		:= FALSE;
			tyP1026McSetTeach.tyMotionStdLifter.tyBtnStop.bRtLk			:= TRUE;

		END_IF

	ELSIF tyP1026McSetTeach.tyMotionStdLifter.tyBtnRst.bRtCompl = TRUE THEN
		tyP1026McSetTeach.tyMotionStdLifter.tyBtnRst.bValue	:= TRUE;
		tyP1026McSetTeach.tyMotionStdLifter.tyBtnRst.bRtLk	:= TRUE;

		eLifterBtmAct	:= LifterActRstAxisErr;

		IF p_eLifterBtmStat = LifterActRstAxisErr AND p_eLifterBtmStatus = Done THEN
			eLifterBtmAct	:= LifterActIdle;

			tyP1026McSetTeach.tyMotionStdLifter.tyBtnRst.bRtCompl	:= FALSE;
			tyP1026McSetTeach.tyMotionStdLifter.tyBtnRst.bValue		:= FALSE;
			tyP1026McSetTeach.tyMotionStdLifter.tyBtnRst.bRtLk		:= FALSE;

			fbLmtRstTm.IN	:= FALSE;
		END_IF

	ELSIF tyP1026McSetTeach.tyTeachLifterPosA.tyBtn2.bRtCompl = TRUE THEN
		tyP1026McSetTeach.tyTeachLifterPosA.tyBtn2.bValue			:= TRUE;
		tyP1026McSetTeach.tyMotionStdLifter.tyBtnStop.bValue		:= FALSE;

		tyP1026McSetTeach.tyTeachLifterPosA.tyBtn2.bRtLk			:= TRUE;
		tyP1026McSetTeach.tyMotionStdLifter.tyBtnStop.bRtLk			:= FALSE;

		diMnlLifterNomSpd	:= tyP1026McSetTeach.tyMotionStdLifter.tyNumNomSpd.diValue;

		eLifterBtmAct	:= LifterActGoAPos;

		IF p_eLifterBtmStat = LifterActGoAPos AND p_eLifterBtmStatus = Done THEN
			eLifterBtmAct	:= LifterActIdle;

			tyP1026McSetTeach.tyTeachLifterPosA.tyBtn2.bRtCompl		:= FALSE;
			tyP1026McSetTeach.tyTeachLifterPosA.tyBtn2.bValue		:= FALSE;
			tyP1026McSetTeach.tyMotionStdLifter.tyBtnStop.bValue	:= TRUE;

			tyP1026McSetTeach.tyTeachLifterPosA.tyBtn2.bRtLk		:= FALSE;
			tyP1026McSetTeach.tyMotionStdLifter.tyBtnStop.bRtLk		:= TRUE;
		END_IF

	ELSIF tyP1026McSetTeach.tyTeachLifterPosB.tyBtn2.bRtCompl = TRUE THEN
		tyP1026McSetTeach.tyTeachLifterPosB.tyBtn2.bValue		:= TRUE;
		tyP1026McSetTeach.tyMotionStdLifter.tyBtnStop.bValue	:= FALSE;

		tyP1026McSetTeach.tyTeachLifterPosB.tyBtn2.bRtLk		:= TRUE;
		tyP1026McSetTeach.tyMotionStdLifter.tyBtnStop.bRtLk		:= FALSE;

		diMnlLifterNomSpd	:= tyP1026McSetTeach.tyMotionStdLifter.tyNumNomSpd.diValue;

		eLifterBtmAct		:= LifterActGoBPos;

		IF p_eLifterBtmStat = LifterActGoBPos AND p_eLifterBtmStatus = Done THEN
			eLifterBtmAct	:= LifterActIdle;

			tyP1026McSetTeach.tyTeachLifterPosB.tyBtn2.bRtCompl		:= FALSE;
			tyP1026McSetTeach.tyTeachLifterPosB.tyBtn2.bValue		:= FALSE;
			tyP1026McSetTeach.tyMotionStdLifter.tyBtnStop.bValue	:= TRUE;

			tyP1026McSetTeach.tyTeachLifterPosB.tyBtn2.bRtLk		:= FALSE;
			tyP1026McSetTeach.tyMotionStdLifter.tyBtnStop.bRtLk		:= TRUE;
		END_IF

	ELSIF tyP1026McSetTeach.tyTeachLifterTopPos.tyBtn2.bRtCompl = TRUE THEN
		tyP1026McSetTeach.tyTeachLifterTopPos.tyBtn2.bValue		:= TRUE;
		tyP1026McSetTeach.tyMotionStdLifter.tyBtnStop.bValue	:= FALSE;

		tyP1026McSetTeach.tyTeachLifterTopPos.tyBtn2.bRtLk		:= TRUE;
		tyP1026McSetTeach.tyMotionStdLifter.tyBtnStop.bRtLk		:= FALSE;

		diMnlLifterNomSpd	:= tyP1026McSetTeach.tyMotionStdLifter.tyNumNomSpd.diValue;

		eLifterBtmAct		:= LifterActGoDPos;

		IF p_eLifterBtmStat = LifterActGoDPos AND p_eLifterBtmStatus = Done THEN
			eLifterBtmAct	:= LifterActIdle;

			tyP1026McSetTeach.tyTeachLifterTopPos.tyBtn2.bRtCompl		:= FALSE;
			tyP1026McSetTeach.tyTeachLifterTopPos.tyBtn2.bValue		:= FALSE;
			tyP1026McSetTeach.tyMotionStdLifter.tyBtnStop.bValue	:= TRUE;

			tyP1026McSetTeach.tyTeachLifterTopPos.tyBtn2.bRtLk		:= FALSE;
			tyP1026McSetTeach.tyMotionStdLifter.tyBtnStop.bRtLk		:= TRUE;
		END_IF

	ELSIF tyP1026McSetTeach.tyTeachLifterBtmPos.tyBtn2.bRtCompl = TRUE THEN
		tyP1026McSetTeach.tyTeachLifterBtmPos.tyBtn2.bValue		:= TRUE;
		tyP1026McSetTeach.tyMotionStdLifter.tyBtnStop.bValue	:= FALSE;

		tyP1026McSetTeach.tyTeachLifterBtmPos.tyBtn2.bRtLk		:= TRUE;
		tyP1026McSetTeach.tyMotionStdLifter.tyBtnStop.bRtLk		:= FALSE;

		diMnlLifterNomSpd	:= tyP1026McSetTeach.tyMotionStdLifter.tyNumNomSpd.diValue;

		eLifterBtmAct		:= LifterActGoEPos;

		IF p_eLifterBtmStat = LifterActGoEPos AND p_eLifterBtmStatus = Done THEN
			eLifterBtmAct	:= LifterActIdle;

			tyP1026McSetTeach.tyTeachLifterBtmPos.tyBtn2.bRtCompl		:= FALSE;
			tyP1026McSetTeach.tyTeachLifterBtmPos.tyBtn2.bValue		:= FALSE;
			tyP1026McSetTeach.tyMotionStdLifter.tyBtnStop.bValue	:= TRUE;

			tyP1026McSetTeach.tyTeachLifterBtmPos.tyBtn2.bRtLk		:= FALSE;
			tyP1026McSetTeach.tyMotionStdLifter.tyBtnStop.bRtLk		:= TRUE;
		END_IF

	ELSIF tyP1026McSetTeach.tyMotionStdLifter.tyBtnMovAbs.bRtCompl = TRUE THEN

		tyP1026McSetTeach.tyMotionStdLifter.tyBtnMovAbs.bValue	:= TRUE;
		tyP1026McSetTeach.tyMotionStdLifter.tyBtnStop.bValue	:= FALSE;

		tyP1026McSetTeach.tyMotionStdLifter.tyBtnMovAbs.bRtLk	:= TRUE;
		tyP1026McSetTeach.tyMotionStdLifter.tyBtnStop.bRtLk		:= FALSE;

		diMnlLifterTargetPos	:= tyP1026McSetTeach.tyMotionStdLifter.tyNumTargetPos.diValue;
		diMnlLifterNomSpd		:= tyP1026McSetTeach.tyMotionStdLifter.tyNumNomSpd.diValue;

		eLifterBtmAct			:= LifterActMovAbs;

		IF p_eLifterBtmStat = LifterActMovAbs AND p_eLifterBtmStatus = Done THEN
			eLifterBtmAct	:= LifterActIdle;

			tyP1026McSetTeach.tyMotionStdLifter.tyBtnMovAbs.bRtCompl	:= FALSE;
			tyP1026McSetTeach.tyMotionStdLifter.tyBtnMovAbs.bValue		:= FALSE;
			tyP1026McSetTeach.tyMotionStdLifter.tyBtnStop.bValue		:= TRUE;

			tyP1026McSetTeach.tyMotionStdLifter.tyBtnMovAbs.bRtLk		:= FALSE;
			tyP1026McSetTeach.tyMotionStdLifter.tyBtnStop.bRtLk			:= TRUE;
		END_IF

	ELSIF tyP1026McSetTeach.tyMotionStdLifter.tyBtnMovRel.bRtCompl = TRUE THEN
		tyP1026McSetTeach.tyMotionStdLifter.tyBtnMovRel.bValue			:= TRUE;
		tyP1026McSetTeach.tyMotionStdLifter.tyBtnStop.bValue			:= FALSE;

		tyP1026McSetTeach.tyMotionStdLifter.tyBtnMovRel.bRtLk			:= TRUE;
		tyP1026McSetTeach.tyMotionStdLifter.tyBtnStop.bRtLk				:= FALSE;

		diMnlLifterStepSize		:= tyP1026McSetTeach.tyMotionStdLifter.tyNumStepSize.diValue;
		diMnlLifterNomSpd		:= tyP1026McSetTeach.tyMotionStdLifter.tyNumNomSpd.diValue;

		eLifterBtmAct		:= LifterActMovRel;

		IF p_eLifterBtmStat = LifterActMovRel AND p_eLifterBtmStatus = Done THEN
			eLifterBtmAct	:= LifterActIdle;

			tyP1026McSetTeach.tyMotionStdLifter.tyBtnMovRel.bRtCompl		:= FALSE;
			tyP1026McSetTeach.tyMotionStdLifter.tyBtnMovRel.bValue			:= FALSE;
			tyP1026McSetTeach.tyMotionStdLifter.tyBtnStop.bValue			:= TRUE;

			tyP1026McSetTeach.tyMotionStdLifter.tyBtnMovRel.bRtLk			:= FALSE;
			tyP1026McSetTeach.tyMotionStdLifter.tyBtnStop.bRtLk				:= TRUE;

		END_IF

	ELSIF (tyP1026McSetTeach.tyMotionStdLifter.tyBtnJogDown.bValue = TRUE) AND (fbJogSlowToFastDlyTm.Q = FALSE) AND (bJogSlow = FALSE) THEN
		tyP1026McSetTeach.tyMotionStdLifter.tyBtnStop.bValue				:= FALSE;
		tyP1026McSetTeach.tyMotionStdLifter.tyBtnStop.bRtLk				:= FALSE;

		fbJogSlowToFastDlyTm.IN		:= TRUE;

		diMnlLifterJogSpd	:= tyP1026McSetTeach.tyMotionStdLifter.tyNumSlwSpd.diValue;

		eLifterBtmAct		:= LifterActJogDown;

		IF p_eLifterBtmStat = LifterActJogDown AND p_eLifterBtmStatus = Done THEN

			eLifterBtmAct	:= LifterActIdle;
			bJogSlow				:= TRUE;

		ELSIF p_eLifterBtmStatus = Error THEN

			fbJogSlowToFastDlyTm.IN	:= FALSE;
			bJogSlow				:= TRUE;

		END_IF

	ELSIF (tyP1026McSetTeach.tyMotionStdLifter.tyBtnJogDown.bValue = TRUE) AND (fbJogSlowToFastDlyTm.Q = TRUE) AND (bJogFast = FALSE) THEN
		tyP1026McSetTeach.tyMotionStdLifter.tyBtnStop.bValue					:= FALSE;
		tyP1026McSetTeach.tyMotionStdLifter.tyBtnStop.bRtLk					:= FALSE;

		fbJogSlowToFastDlyTm.IN		:= TRUE;

		diMnlLifterJogSpd	:= tyP1026McSetTeach.tyMotionStdLifter.tyNumNomSpd.diValue;

		eLifterBtmAct		:= LifterActJogDown;

		IF p_eLifterBtmStat = LifterActJogDown AND p_eLifterBtmStatus = Done THEN
			eLifterBtmAct	:= LifterActIdle;
			bJogFast				:= TRUE;
		ELSIF p_eLifterBtmStatus = Error THEN
			fbJogSlowToFastDlyTm.IN	:= FALSE;
			bJogFast				:= TRUE;
		END_IF

	ELSIF (tyP1026McSetTeach.tyMotionStdLifter.tyBtnJogUp.bValue = TRUE) AND (fbJogSlowToFastDlyTm.Q = FALSE) AND (bJogSlow = FALSE) THEN
		tyP1026McSetTeach.tyMotionStdLifter.tyBtnStop.bValue				:= FALSE;
		tyP1026McSetTeach.tyMotionStdLifter.tyBtnStop.bRtLk				:= FALSE;

		fbJogSlowToFastDlyTm.IN		:= TRUE;

		diMnlLifterJogSpd	:= tyP1026McSetTeach.tyMotionStdLifter.tyNumSlwSpd.diValue;

		eLifterBtmAct		:= LifterActJogUp;

		IF p_eLifterBtmStat = LifterActJogUp AND p_eLifterBtmStatus = Done THEN
			eLifterBtmAct	:= LifterActIdle;
			bJogSlow				:= TRUE;

		ELSIF p_eLifterBtmStatus = Error THEN
			fbJogSlowToFastDlyTm.IN	:= FALSE;
			bJogSlow				:= TRUE;
		END_IF

	ELSIF (tyP1026McSetTeach.tyMotionStdLifter.tyBtnJogUp.bValue = TRUE) AND (fbJogSlowToFastDlyTm.Q = TRUE) AND (bJogFast = FALSE) THEN

		tyP1026McSetTeach.tyMotionStdLifter.tyBtnStop.bValue				:= FALSE;
		tyP1026McSetTeach.tyMotionStdLifter.tyBtnStop.bRtLk					:= FALSE;

		fbJogSlowToFastDlyTm.IN		:= TRUE;

		diMnlLifterJogSpd	:= tyP1026McSetTeach.tyMotionStdLifter.tyNumNomSpd.diValue;

		eLifterBtmAct		:= LifterActJogUp;

		IF p_eLifterBtmStat = LifterActJogUp AND p_eLifterBtmStatus = Done THEN
			eLifterBtmAct	:= LifterActIdle;
			bJogFast	:= TRUE;

		ELSIF p_eLifterBtmStatus = Error THEN
			fbJogSlowToFastDlyTm.IN	:= FALSE;
			bJogFast				:= TRUE;
		END_IF
	END_IF

	IF tyP1026McSetTeach.tyInOutletShutterFB.tyBtnOpen.bRtCompl = TRUE THEN
		tyP1026McSetTeach.tyInOutletShutterFB.tyBtnOpen.bRtCompl	:= FALSE;

		tyP1026McSetTeach.tyInOutletShutterFB.tyBtnOpen.bValue	:= TRUE;
		tyP1026McSetTeach.tyInOutletShutterFB.tyBtnClose.bValue	:= FALSE;

	ELSIF tyP1026McSetTeach.tyInOutletShutterFB.tyBtnClose.bRtCompl = TRUE THEN
		tyP1026McSetTeach.tyInOutletShutterFB.tyBtnClose.bRtCompl	:= FALSE;

		tyP1026McSetTeach.tyInOutletShutterFB.tyBtnClose.bValue	:= TRUE;
		tyP1026McSetTeach.tyInOutletShutterFB.tyBtnOpen.bValue	:= FALSE;
	END_IF

	IF tyP1026McSetTeach.tyInOutletShutterFB.tyBtnOpen.bValue = TRUE THEN
		eInShutterAct	:= PneuActRet;
		eOutShutterAct	:= PneuActRet;
		eOutShutterAct2	:= PneuActRet;
		eOutShutterAct3	:= PneuActRet;

		IF (p_eInShutterStat = PneuActRet AND p_eInShutterStatus = Done)
			AND (p_eOutShutterStat = PneuActRet AND p_eOutShutterStatus = Done)
			AND (p_eOutShutterStat2 = PneuActRet AND p_eOutShutterStatus2 = Done)
			AND (p_eOutShutterStat3 = PneuActRet AND p_eOutShutterStatus3 = Done)
			THEN
			eInShutterAct	:= PneuActIdle;
			eOutShutterAct	:= PneuActIdle;
			eOutShutterAct2	:= PneuActIdle;
			eOutShutterAct3	:= PneuActIdle;
			tyP1026McSetTeach.tyInOutletShutterFB.tyBtnOpen.bValue	:= FALSE;
		ELSIF p_eInShutterStatus = Error OR p_eOutShutterStatus = Error OR p_eOutShutterStatus2 = Error OR p_eOutShutterStatus3 = Error THEN
			tyP1026McSetTeach.tyInOutletShutterFB.tyBtnOpen.bValue	:= FALSE;
		END_IF

	ELSIF tyP1026McSetTeach.tyInOutletShutterFB.tyBtnClose.bValue = TRUE THEN
		eInShutterAct	:= PneuActExt;
		eOutShutterAct	:= PneuActExt;
		eOutShutterAct2	:= PneuActExt;
		eOutShutterAct3	:= PneuActExt;
		IF (p_eInShutterStat = PneuActExt AND p_eInShutterStatus = Done)
			AND (p_eOutShutterStat = PneuActExt AND p_eOutShutterStatus = Done)
			AND (p_eOutShutterStat2 = PneuActExt AND p_eOutShutterStatus2 = Done)
			AND (p_eOutShutterStat3 = PneuActExt AND p_eOutShutterStatus3 = Done)
			THEN
			eInShutterAct	:= PneuActIdle;
			eOutShutterAct	:= PneuActIdle;
			eOutShutterAct2	:= PneuActIdle;
			eOutShutterAct3	:= PneuActIdle;
			tyP1026McSetTeach.tyInOutletShutterFB.tyBtnClose.bValue := FALSE;
		ELSIF p_eInShutterStatus = Error OR p_eOutShutterStatus = Error OR p_eOutShutterStatus2 = Error OR p_eOutShutterStatus3 = Error THEN
			tyP1026McSetTeach.tyInOutletShutterFB.tyBtnClose.bValue := FALSE;
		END_IF
	END_IF

	IF p_eLifterBtmStat = LifterActStop AND (p_eLifterBtmStatus = Done OR p_eLifterBtmStatus = Error) THEN
		eLifterBtmAct	:= LifterActIdle;
	END_IF

	//bypass curtain sensor
	IF bTeachLifterPosA OR bTeachLifterPosB THEN
		bBypCurtainSen			:= tyP1026McSetTeach.tyTeachLifterPosA.tyBtn4.bValue OR tyP1026McSetTeach.tyTeachLifterPosB.tyBtn4.bValue;
		bBypCurtainPBLED		:= tyP1026McSetTeach.tyTeachLifterPosA.tyBtn4.bValue OR tyP1026McSetTeach.tyTeachLifterPosB.tyBtn4.bValue;
	END_IF

END_ACTION
```

#### Act_OptP1026LifterFBStat.st
```iecst
ACTION Act_OptP1026LifterFBStat:

	IF p_bLifterBtmAxisErr = TRUE THEN
		tyP1026McSetTeach.tyMotionStdLifter.tyStringStat.sValue		:= p_sLifterBtmAxisErrTxt;
	ELSE
		tyP1026McSetTeach.tyMotionStdLifter.tyStringStat.sValue		:= p_sLifterBtmStatTxt;
	END_IF

END_ACTION
```

#### Act_OptP1026LifterMask.st
```iecst
ACTION Act_OptP1026LifterMask:

	// Interlock Power
	IF p_bLifterBtmAxisErr = TRUE AND p_bLifterBtmPwrOn = FALSE THEN
		fUIInRtStatOff(ADR(tyP1026McSetTeach.tyMotionStdLifter.tyBtnPwr.uiMaskRtStat));
		tyP1026McSetTeach.tyMotionStdLifter.tyBtnPwr.bValue		:= FALSE;
	ELSE
		fUIInRtStatHide(ADR(tyP1026McSetTeach.tyMotionStdLifter.tyBtnPwr.uiMaskRtStat));
	END_IF

	// Interlock Others Move
	IF p_bLifterBtmAxisErr = TRUE OR p_bLifterBtmPwrOn = FALSE THEN
		fUIInRtStatOff(ADR(tyP1026McSetTeach.tyMotionStdLifter.tyBtnOrigin.uiMaskRtStat));
		fUIInRtStatOff(ADR(tyP1026McSetTeach.tyMotionStdLifter.tyBtnMovRel.uiMaskRtStat));
		fUIInRtStatOff(ADR(tyP1026McSetTeach.tyMotionStdLifter.tyBtnJogUp.uiMaskRtStat));
		fUIInRtStatOff(ADR(tyP1026McSetTeach.tyMotionStdLifter.tyBtnJogDown.uiMaskRtStat));
	ELSE
		fUIInRtStatHide(ADR(tyP1026McSetTeach.tyMotionStdLifter.tyBtnOrigin.uiMaskRtStat));
		fUIInRtStatHide(ADR(tyP1026McSetTeach.tyMotionStdLifter.tyBtnMovRel.uiMaskRtStat));
		fUIInRtStatHide(ADR(tyP1026McSetTeach.tyMotionStdLifter.tyBtnJogUp.uiMaskRtStat));
		fUIInRtStatHide(ADR(tyP1026McSetTeach.tyMotionStdLifter.tyBtnJogDown.uiMaskRtStat));
	END_IF

	// Interlock Move Absolute
	IF p_bLifterBtmAxisErr = TRUE OR p_bLifterBtmPwrOn = FALSE OR p_bLifterBtmIsHomed = FALSE THEN

		fUIInRtStatOff(ADR(tyP1026McSetTeach.tyTeachLifterPosA.tyBtn2.uiMaskRtStat));
		fUIInRtStatOff(ADR(tyP1026McSetTeach.tyTeachLifterPosB.tyBtn2.uiMaskRtStat));
		fUIInRtStatOff(ADR(tyP1026McSetTeach.tyMotionStdLifter.tyBtnMovAbs.uiMaskRtStat));
	ELSE
		fUIInRtStatHide(ADR(tyP1026McSetTeach.tyTeachLifterPosA.tyBtn2.uiMaskRtStat));
		fUIInRtStatHide(ADR(tyP1026McSetTeach.tyTeachLifterPosB.tyBtn2.uiMaskRtStat));
		fUIInRtStatHide(ADR(tyP1026McSetTeach.tyMotionStdLifter.tyBtnMovAbs.uiMaskRtStat));
	END_IF

	//Interlock Limit Sensor
	IF tyP1026McSetTeach.tyMotionStdLifter.tyBtnDownLmtSen.bValue = TRUE THEN
		fUIInRtStatOff(ADR(tyP1026McSetTeach.tyMotionStdLifter.tyBtnJogDown.uiMaskRtStat));
	END_IF

	IF tyP1026McSetTeach.tyMotionStdLifter.tyBtnUpLmtSen.bValue = TRUE THEN
		fUIInRtStatOff(ADR(tyP1026McSetTeach.tyMotionStdLifter.tyBtnJogUp.uiMaskRtStat));
	END_IF

	// Interlock When Moving
	IF tyP1026McSetTeach.tyMotionStdLifter.tyBtnOrigin.bRtCompl = TRUE THEN
		fUIInRtStatOff(ADR(tyP1026McSetTeach.tyMotionStdLifter.tyBtnMovAbs.uiMaskRtStat));
		fUIInRtStatOff(ADR(tyP1026McSetTeach.tyMotionStdLifter.tyBtnMovRel.uiMaskRtStat));
		fUIInRtStatOff(ADR(tyP1026McSetTeach.tyMotionStdLifter.tyBtnJogUp.uiMaskRtStat));
		fUIInRtStatOff(ADR(tyP1026McSetTeach.tyMotionStdLifter.tyBtnJogDown.uiMaskRtStat));

		fUIInRtStatOff(ADR(tyP1026McSetTeach.tyTeachLifterPosA.tyBtn2.uiMaskRtStat));
		fUIInRtStatOff(ADR(tyP1026McSetTeach.tyTeachLifterPosB.tyBtn2.uiMaskRtStat));

	ELSIF tyP1026McSetTeach.tyMotionStdLifter.tyBtnMovAbs.bRtCompl = TRUE THEN
		fUIInRtStatOff(ADR(tyP1026McSetTeach.tyMotionStdLifter.tyBtnOrigin.uiMaskRtStat));
		fUIInRtStatOff(ADR(tyP1026McSetTeach.tyMotionStdLifter.tyBtnMovRel.uiMaskRtStat));
		fUIInRtStatOff(ADR(tyP1026McSetTeach.tyMotionStdLifter.tyBtnJogUp.uiMaskRtStat));
		fUIInRtStatOff(ADR(tyP1026McSetTeach.tyMotionStdLifter.tyBtnJogDown.uiMaskRtStat));

		fUIInRtStatOff(ADR(tyP1026McSetTeach.tyTeachLifterPosA.tyBtn2.uiMaskRtStat));
		fUIInRtStatOff(ADR(tyP1026McSetTeach.tyTeachLifterPosB.tyBtn2.uiMaskRtStat));

	ELSIF tyP1026McSetTeach.tyMotionStdLifter.tyBtnMovRel.bRtCompl = TRUE THEN
		fUIInRtStatOff(ADR(tyP1026McSetTeach.tyMotionStdLifter.tyBtnOrigin.uiMaskRtStat));
		fUIInRtStatOff(ADR(tyP1026McSetTeach.tyMotionStdLifter.tyBtnMovAbs.uiMaskRtStat));
		fUIInRtStatOff(ADR(tyP1026McSetTeach.tyMotionStdLifter.tyBtnJogUp.uiMaskRtStat));
		fUIInRtStatOff(ADR(tyP1026McSetTeach.tyMotionStdLifter.tyBtnJogDown.uiMaskRtStat));

		fUIInRtStatOff(ADR(tyP1026McSetTeach.tyTeachLifterPosA.tyBtn2.uiMaskRtStat));
		fUIInRtStatOff(ADR(tyP1026McSetTeach.tyTeachLifterPosB.tyBtn2.uiMaskRtStat));

	ELSIF tyP1026McSetTeach.tyMotionStdLifter.tyBtnJogDown.bRtCompl = TRUE OR tyP1026McSetTeach.tyMotionStdLifter.tyBtnJogDown.bValue = TRUE THEN
		fUIInRtStatOff(ADR(tyP1026McSetTeach.tyMotionStdLifter.tyBtnOrigin.uiMaskRtStat));
		fUIInRtStatOff(ADR(tyP1026McSetTeach.tyMotionStdLifter.tyBtnMovAbs.uiMaskRtStat));
		fUIInRtStatOff(ADR(tyP1026McSetTeach.tyMotionStdLifter.tyBtnMovRel.uiMaskRtStat));
		fUIInRtStatOff(ADR(tyP1026McSetTeach.tyMotionStdLifter.tyBtnJogUp.uiMaskRtStat));

		fUIInRtStatOff(ADR(tyP1026McSetTeach.tyTeachLifterPosA.tyBtn2.uiMaskRtStat));
		fUIInRtStatOff(ADR(tyP1026McSetTeach.tyTeachLifterPosB.tyBtn2.uiMaskRtStat));

	ELSIF tyP1026McSetTeach.tyMotionStdLifter.tyBtnJogUp.bRtCompl = TRUE OR tyP1026McSetTeach.tyMotionStdLifter.tyBtnJogUp.bValue = TRUE THEN
		fUIInRtStatOff(ADR(tyP1026McSetTeach.tyMotionStdLifter.tyBtnOrigin.uiMaskRtStat));
		fUIInRtStatOff(ADR(tyP1026McSetTeach.tyMotionStdLifter.tyBtnMovAbs.uiMaskRtStat));
		fUIInRtStatOff(ADR(tyP1026McSetTeach.tyMotionStdLifter.tyBtnMovRel.uiMaskRtStat));
		fUIInRtStatOff(ADR(tyP1026McSetTeach.tyMotionStdLifter.tyBtnJogDown.uiMaskRtStat));

		fUIInRtStatOff(ADR(tyP1026McSetTeach.tyTeachLifterPosA.tyBtn2.uiMaskRtStat));
		fUIInRtStatOff(ADR(tyP1026McSetTeach.tyTeachLifterPosB.tyBtn2.uiMaskRtStat));

	ELSIF tyP1026McSetTeach.tyTeachLifterPosA.tyBtn2.bRtCompl = TRUE THEN
		fUIInRtStatOff(ADR(tyP1026McSetTeach.tyMotionStdLifter.tyBtnOrigin.uiMaskRtStat));
		fUIInRtStatOff(ADR(tyP1026McSetTeach.tyMotionStdLifter.tyBtnMovAbs.uiMaskRtStat));
		fUIInRtStatOff(ADR(tyP1026McSetTeach.tyMotionStdLifter.tyBtnMovRel.uiMaskRtStat));
		fUIInRtStatOff(ADR(tyP1026McSetTeach.tyMotionStdLifter.tyBtnJogUp.uiMaskRtStat));
		fUIInRtStatOff(ADR(tyP1026McSetTeach.tyMotionStdLifter.tyBtnJogDown.uiMaskRtStat));

	ELSIF tyP1026McSetTeach.tyTeachLifterPosB.tyBtn2.bRtCompl = TRUE THEN
		fUIInRtStatOff(ADR(tyP1026McSetTeach.tyMotionStdLifter.tyBtnOrigin.uiMaskRtStat));
		fUIInRtStatOff(ADR(tyP1026McSetTeach.tyMotionStdLifter.tyBtnMovAbs.uiMaskRtStat));
		fUIInRtStatOff(ADR(tyP1026McSetTeach.tyMotionStdLifter.tyBtnMovRel.uiMaskRtStat));
		fUIInRtStatOff(ADR(tyP1026McSetTeach.tyMotionStdLifter.tyBtnJogUp.uiMaskRtStat));
		fUIInRtStatOff(ADR(tyP1026McSetTeach.tyMotionStdLifter.tyBtnJogDown.uiMaskRtStat));

	END_IF

	//Axis Error
	IF tyP1026McSetTeach.tyMotionStdLifter.tyBtnPwr.bRtCompl = TRUE THEN
		fUIInRtStatOff(ADR(tyP1026McSetTeach.tyMotionStdLifter.tyBtnRst.uiMaskRtStat));
	ELSE
		fUIInRtStatHide(ADR(tyP1026McSetTeach.tyMotionStdLifter.tyBtnRst.uiMaskRtStat));
	END_IF

	//Interlock Button Get
	IF p_bLifterBtmAxisErr = TRUE OR p_bLifterBtmIsHomed = FALSE OR p_bLifterBtmFwdLmtSen = TRUE OR p_bLifterBtmRevLmtSen = TRUE THEN
		fUIInRtStatOff(ADR(tyP1026McSetTeach.tyTeachLifterPosA.tyBtn1.uiMaskRtStat));
		fUIInRtStatOff(ADR(tyP1026McSetTeach.tyTeachLifterPosB.tyBtn1.uiMaskRtStat));
	ELSE
		fUIInRtStatHide(ADR(tyP1026McSetTeach.tyTeachLifterPosA.tyBtn1.uiMaskRtStat));
		fUIInRtStatHide(ADR(tyP1026McSetTeach.tyTeachLifterPosB.tyBtn1.uiMaskRtStat));
	END_IF

END_ACTION
```

#### Act_OptP1026LifterUpdtDat.st
```iecst
ACTION Act_OptP1026LifterUpdtDat:

	tyP1026McSetTeach.tyMotionStdLifter.tyNumCurrPos.diValue		:= p_diLifterBtmActualPos;
	tyP1026McSetTeach.tyMotionStdLifter.tyNumErrCode.diValue		:= UDINT_TO_DINT(p_udiLifterBtmAxisErrID);
	tyP1026McSetTeach.tyMotionStdLifter.tyBitmapPwr.usiValueIdx		:= BOOL_TO_USINT(p_bLifterBtmPwrOn);
	tyP1026McSetTeach.tyMotionStdLifter.tyBitmapRst.usiValueIdx		:= BOOL_TO_USINT(NOT p_bLifterBtmAxisErr);
	tyP1026McSetTeach.tyMotionStdLifter.tyBitmapOrigin.usiValueIdx	:= BOOL_TO_USINT(p_bLifterBtmIsHomed);
	tyP1026McSetTeach.tyMotionStdLifter.tyBtnUpLmtSen.bValue		:= p_bLifterBtmUpSen;
	tyP1026McSetTeach.tyMotionStdLifter.tyBtnDownLmtSen.bValue		:= p_bLifterBtmDownSen;

	//Machine Bitmap
	IF p_bLifterBtmIsHomed = TRUE THEN
		IF p_diLifterBtmActualPos <= (p_tyNtParamCurr.tyUILifterTargetPos.diMax / 3) THEN
			tyP1026McSetTeach.tyMotionStdLifter.tyBitmapMc.uiValueIdx 	:= 2;
		ELSIF p_diLifterBtmActualPos <= (p_tyNtParamCurr.tyUILifterTargetPos.diMax / 3 * 2) THEN
			tyP1026McSetTeach.tyMotionStdLifter.tyBitmapMc.uiValueIdx 	:= 3;
		ELSE
			tyP1026McSetTeach.tyMotionStdLifter.tyBitmapMc.uiValueIdx 	:= 4;
		END_IF
	ELSE
		tyP1026McSetTeach.tyMotionStdLifter.tyBitmapMc.uiValueIdx	:= 2;
	END_IF

	IF p_tyNtParamCurr.eProjMag = ULMagDual THEN
		IF p_tyNtParamCurr.bProjLifterMagPlatform AND p_tyNtParamCurr.bUIConvDirRL THEN
			IF 	tyP1026McSetTeach.tyMotionStdLifter.tyBitmapMc.uiValueIdx < 700 THEN
				tyP1026McSetTeach.tyMotionStdLifter.tyBitmapMc.uiValueIdx	:= tyP1026McSetTeach.tyMotionStdLifter.tyBitmapMc.uiValueIdx + 700;
			END_IF
		ELSIF p_tyNtParamCurr.bProjLifterMagPlatform THEN
			IF p_tyNtParamCurr.bProjMagConvLane1Prep = FALSE THEN
				IF 	tyP1026McSetTeach.tyMotionStdLifter.tyBitmapMc.uiValueIdx < 600 THEN
					tyP1026McSetTeach.tyMotionStdLifter.tyBitmapMc.uiValueIdx	:= tyP1026McSetTeach.tyMotionStdLifter.tyBitmapMc.uiValueIdx + 600;
				END_IF
			ELSE
				IF 	tyP1026McSetTeach.tyMotionStdLifter.tyBitmapMc.uiValueIdx < 900 THEN
					tyP1026McSetTeach.tyMotionStdLifter.tyBitmapMc.uiValueIdx	:= tyP1026McSetTeach.tyMotionStdLifter.tyBitmapMc.uiValueIdx + 900;
				END_IF
			END_IF
		ELSIF p_tyNtParamCurr.bMagAutoVerifyPrep = FALSE THEN
			IF 	tyP1026McSetTeach.tyMotionStdLifter.tyBitmapMc.uiValueIdx < 100 THEN
				tyP1026McSetTeach.tyMotionStdLifter.tyBitmapMc.uiValueIdx	:= tyP1026McSetTeach.tyMotionStdLifter.tyBitmapMc.uiValueIdx + 300;
			END_IF
		ELSE
			IF 	tyP1026McSetTeach.tyMotionStdLifter.tyBitmapMc.uiValueIdx < 300 THEN
				tyP1026McSetTeach.tyMotionStdLifter.tyBitmapMc.uiValueIdx	:= tyP1026McSetTeach.tyMotionStdLifter.tyBitmapMc.uiValueIdx + 300;
			END_IF
		END_IF
	ELSIF p_tyNtParamCurr.eProjMag = ULMagTriple THEN
		IF p_tyNtParamCurr.bProjLifterMagPlatform AND p_tyNtParamCurr.bUIConvDirRL THEN
			IF 	tyP1026McSetTeach.tyMotionStdLifter.tyBitmapMc.uiValueIdx < 800 THEN
				tyP1026McSetTeach.tyMotionStdLifter.tyBitmapMc.uiValueIdx	:= tyP1026McSetTeach.tyMotionStdLifter.tyBitmapMc.uiValueIdx + 800;
			END_IF
		ELSIF p_tyNtParamCurr.bProjLifterMagPlatform THEN
			IF 	tyP1026McSetTeach.tyMotionStdLifter.tyBitmapMc.uiValueIdx < 500 THEN
				tyP1026McSetTeach.tyMotionStdLifter.tyBitmapMc.uiValueIdx	:= tyP1026McSetTeach.tyMotionStdLifter.tyBitmapMc.uiValueIdx + 500;
			END_IF
		ELSIF p_tyNtParamCurr.bMagAutoVerifyPrep = TRUE AND p_tyNtParamCurr.bProjMotorizedPusherPrep = FALSE THEN
			IF 	tyP1026McSetTeach.tyMotionStdLifter.tyBitmapMc.uiValueIdx < 200 THEN
				tyP1026McSetTeach.tyMotionStdLifter.tyBitmapMc.uiValueIdx	:= tyP1026McSetTeach.tyMotionStdLifter.tyBitmapMc.uiValueIdx + 200;
			END_IF
		ELSIF p_tyNtParamCurr.bMagAutoVerifyPrep = FALSE AND p_tyNtParamCurr.bProjMotorizedPusherPrep = TRUE THEN
			IF 	tyP1026McSetTeach.tyMotionStdLifter.tyBitmapMc.uiValueIdx < 400 THEN
				tyP1026McSetTeach.tyMotionStdLifter.tyBitmapMc.uiValueIdx	:= tyP1026McSetTeach.tyMotionStdLifter.tyBitmapMc.uiValueIdx + 400;
			END_IF
		END_IF
	END_IF

END_ACTION
```
